      _stMsg.eType                  := E_MessageType.eMessageError;
      _stMsg.eDevice                := e_Device.Axis + TO_DINT(_AxisRef.NcToPlc.AxisId);
      _stMsg.eSubdevice             := e_Subdevice.fbCoeRead;

      _stMsg.iErrorNumber           := SEL((_fbCoeRead.CANopenErrId > 0), _fbCoeRead.AdsErrId, _fbCoeRead.CANopenErrId);

      _stMsg.sText                  := TO_STRING(_eState);
      f_MessageSet(_stMsg);

      _fbCoeRead(
                Execute             := FALSE,
                NetId               := _AxisRef.ADS.NetId, 
                Axis                := _AxisRef);

    ELSIF NOT _fbCoeRead.Busy
    THEN
      _eState                       := E_PROGRESS.WORKING;
    END_IF
*)
END_CASE
CASE _eState
OF
  E_PROGRESS.PROGRESS_WORKING:
    _eState                         := E_PROGRESS.PROGRESS_DONE;
    // set default for axis release
    AxisEnableNegative              := TRUE;
    AxisEnablePositive              := TRUE;

    // clear fb
    _fbCoeRead(
              Execute               := FALSE,
              NetId                 := _AxisRef.ADS.NetId, 
              Axis                  := _AxisRef);

    _stMsg.eType                    := E_MessageType.eMessageInfo;
    _stMsg.eDevice                  := e_Device.Axis + (_AxisRef.NcToPlc.AxisId);
    _stMsg.eSubdevice               := e_Subdevice.AxisStartUp;
    _stMsg.iErrorNumber             := 0;
    _stMsg.sText                    := concat('Axis Init: ', _sDeviceName);
    _stMsg.sText                    := concat(_stMsg.sText, ' : ');
    _stMsg.sText                    := concat(_stMsg.sText, TO_STRING(_eState));

  IF (_MessageLevel > E_MessageType.eMessageError)
  THEN
    f_MessageSet(_stMsg);
  END_IF
END_CASE

AxisInit                            := _eState;
END_METHOD

METHOD AxisMoveToPosition : E_PROGRESS
VAR_INPUT
  Execute           : BOOL;
  Data              : ST_MOVE_DATA;
END_VAR
VAR_INST
  _eres,
  _eState           : E_PROGRESS;
END_VAR
IF NOT Check() THEN AxisMoveToPosition := E_PROGRESS.PROGRESS_ERROR; RETURN; END_IF
IF NOT Execute THEN _eState := E_PROGRESS.PROGRESS_INIT; END_IF

CASE _eState
OF
  E_PROGRESS.PROGRESS_INIT:
    IF Execute 
    THEN
      _eState               := E_PROGRESS.PROGRESS_BUSY;
    END_IF
END_CASE
CASE _eState
OF
  E_PROGRESS.PROGRESS_BUSY:
    _eState                 := E_PROGRESS.PROGRESS_OCCUPIED;
    _eres                   := MoveToPos(
                                      Execute    := FALSE, 
                                      Position   := Data.rSetPos, 
                                      Vel        := Data.rSetVelo, 
                                      Acc        := Data.rAcc, 
                                      Dec        := Data.rDec, 
                                      Jerk       := Data.rJerk, 
                                      BufferMode := Tc2_MC2.MC_BufferMode.MC_Aborting);
END_CASE
CASE _eState
OF
  E_PROGRESS.PROGRESS_OCCUPIED:
    _eres                   := MoveToPos(
                                      Execute    := TRUE, 
                                      Position   := Data.rSetPos, 
                                      Vel        := Data.rSetVelo, 
                                      Acc        := Data.rAcc, 
                                      Dec        := Data.rDec, 
                                      Jerk       := Data.rJerk, 
                                      BufferMode := Tc2_MC2.MC_BufferMode.MC_Aborting);

    IF (_eres = E_PROGRESS.PROGRESS_ERROR)
    THEN
        _eState             := E_PROGRESS.PROGRESS_ERROR;
    ELSIF (_eres = E_PROGRESS.PROGRESS_DONE)
    THEN 
      _eState               := E_PROGRESS.PROGRESS_WORKING;
    END_IF
END_CASE
CASE _eState
OF
  E_PROGRESS.PROGRESS_WORKING:
    _eState                 := E_PROGRESS.PROGRESS_DONE;
    _eres                   := MoveToPos(
                                      Execute    := FALSE, 
                                      Position   := Data.rSetPos, 
                                      Vel        := Data.rSetVelo, 
                                      Acc        := Data.rAcc, 
                                      Dec        := Data.rDec, 
                                      Jerk       := Data.rJerk, 
                                      BufferMode := Tc2_MC2.MC_BufferMode.MC_Aborting);
END_CASE

AxisMoveToPosition := _eState;
END_METHOD

METHOD AxisMoveVelocity : E_PROGRESS
VAR_INPUT
  Execute           : BOOL;
  Data              : ST_MOVE_DATA;
END_VAR
VAR_INST
  _eres,
  _eState           : E_PROGRESS;
END_VAR
IF NOT Check() THEN AxisMoveVelocity := E_PROGRESS.PROGRESS_ERROR; RETURN; END_IF
IF NOT Execute THEN _eState := E_PROGRESS.PROGRESS_INIT; END_IF

CASE _eState
OF
  E_PROGRESS.PROGRESS_INIT:
    IF Execute 
    THEN
      _eState               := E_PROGRESS.PROGRESS_BUSY;
    END_IF
END_CASE
CASE _eState
OF
  E_PROGRESS.PROGRESS_BUSY:
    _eState                 := E_PROGRESS.PROGRESS_OCCUPIED;
    _eres                   := MoveVelo(
                                    Execute     := FALSE, 
                                    Velocity    := Data.rSetVelo, 
                                    Acc         := Data.rAcc, 
                                    Dec         := Data.rDec, 
                                    Jerk        := Data.rJerk, 
                                    Direction   := Data.iDirection, 
                                    BufferMode  := Tc2_MC2.MC_BufferMode.MC_Aborting);
END_CASE
CASE _eState
OF
  E_PROGRESS.PROGRESS_OCCUPIED:
    _eres                   := MoveVelo(
                                    Execute     := TRUE, 
                                    Velocity    := Data.rSetVelo, 
                                    Acc         := Data.rAcc, 
                                    Dec         := Data.rDec, 
                                    Jerk        := Data.rJerk, 
                                    Direction   := Data.iDirection, 
                                    BufferMode  := Tc2_MC2.MC_BufferMode.MC_Aborting);
    IF (_eres = E_PROGRESS.PROGRESS_ERROR)
    THEN
        _eState             := E_PROGRESS.PROGRESS_ERROR;
    ELSIF (_eres = E_PROGRESS.PROGRESS_DONE)
    THEN 
      _eState               := E_PROGRESS.PROGRESS_WORKING;
    END_IF
END_CASE
CASE _eState
OF
  E_PROGRESS.PROGRESS_WORKING:
    _eState                 := E_PROGRESS.PROGRESS_DONE;
    _eres                   := MoveVelo(
                                    Execute     := FALSE, 
                                    Velocity    := Data.rSetVelo, 
                                    Acc         := Data.rAcc, 
                                    Dec         := Data.rDec, 
                                    Jerk        := Data.rJerk, 
                                    Direction   := Data.iDirection, 
                                    BufferMode  := Tc2_MC2.MC_BufferMode.MC_Aborting);
END_CASE

AxisMoveVelocity                := _eState;
END_METHOD

METHOD AxisParameterRead : E_PROGRESS
VAR_INPUT
  Execute           : BOOL;
  ParameterNr       : Tc2_MC2.MC_AxisParameter;
END_VAR
VAR_INST
  _eres,
  _eState           : E_PROGRESS;
  _rValue           : LREAL;
END_VAR
IF NOT Check() THEN AxisParameterRead := E_PROGRESS.PROGRESS_ERROR; RETURN; END_IF
IF NOT Execute THEN _eState := E_PROGRESS.PROGRESS_INIT; END_IF

CASE _eState
OF
  E_PROGRESS.PROGRESS_INIT:
    IF Execute 
    THEN
      _rValue                                     := 0.0;
      _eState                                     := E_PROGRESS.PROGRESS_BUSY;
    END_IF
END_CASE
CASE _eState
OF
  E_PROGRESS.PROGRESS_BUSY:
    _eState                                       := E_PROGRESS.PROGRESS_OCCUPIED;
    _eres           := ReadParameter(
                                  Execute         := FALSE,
                                  ParameterNumber := ParameterNr);
END_CASE
CASE _eState
OF
  E_PROGRESS.PROGRESS_OCCUPIED:
    _eres           := ReadParameter(
                                  Execute         := TRUE,
                                  ParameterNumber := ParameterNr);

    IF (_eres = E_PROGRESS.PROGRESS_ERROR)
    THEN
      _eState                                     := E_PROGRESS.PROGRESS_ERROR;
    ELSIF (_eres = E_PROGRESS.PROGRESS_DONE)
    THEN 
      _eState                                     := E_PROGRESS.PROGRESS_WORKING;
    END_IF

  E_PROGRESS.PROGRESS_WORKING:
    _eState                                       := E_PROGRESS.PROGRESS_DONE;
    _eres           := ReadParameter(
                                  Execute         := FALSE,
                                  ParameterNumber := ParameterNr);

    _NcParameterWrt^[_nAxisIndex].rValue          :=
    _rParameterReadValue                          := 
    _rValue                                       :=ReadParameterValue;
END_CASE

AxisParameterRead := _eState;
END_METHOD

METHOD AxisParameterWrite : E_PROGRESS
VAR_INPUT
  Execute           : BOOL;
  ParameterNr       : Tc2_MC2.MC_AxisParameter;
END_VAR
VAR_INST
  _eres,
  _eState           : E_PROGRESS;
  _rValue           : LREAL;
END_VAR
IF NOT Check() THEN AxisParameterWrite := E_PROGRESS.PROGRESS_ERROR; RETURN; END_IF
IF NOT Execute THEN _eState := E_PROGRESS.PROGRESS_INIT; END_IF

CASE _eState
OF
  E_PROGRESS.PROGRESS_INIT:
    IF Execute 
    THEN
      _rValue                                     := _NcParameterWrt^[_nAxisIndex].rValue;
      _eState                                     := E_PROGRESS.PROGRESS_BUSY;
    END_IF
END_CASE
CASE _eState
OF
  E_PROGRESS.PROGRESS_BUSY:
    _eState                                       := E_PROGRESS.PROGRESS_OCCUPIED;
    _eres           := WriteParameter(
                                  Execute         := FALSE,
                                  Value           := _rValue,
                                  ParameterNumber := ParameterNr);
END_CASE
CASE _eState
OF
  E_PROGRESS.PROGRESS_OCCUPIED:
    _eres           := WriteParameter(
                                  Execute         := TRUE,
                                  Value           := _rValue,
                                  ParameterNumber := ParameterNr);
    IF (_eres = E_PROGRESS.PROGRESS_ERROR)
    THEN
      _eState                                     := E_PROGRESS.PROGRESS_ERROR;
    ELSIF (_eres = E_PROGRESS.PROGRESS_DONE)
    THEN 
      _eState                                     := E_PROGRESS.PROGRESS_WORKING;
    END_IF

  E_PROGRESS.PROGRESS_WORKING:
    _eState                                       := E_PROGRESS.PROGRESS_DONE;
    _eres           := WriteParameter(
                                  Execute         := FALSE,
                                  Value           := _rValue,
                                  ParameterNumber := ParameterNr);
END_CASE

AxisParameterWrite                                    := _eState;
END_METHOD

METHOD AxisParameterWritePersistent : E_PROGRESS
VAR_INPUT
  Execute           : BOOL;
  ParameterNr       : Tc2_MC2.MC_AxisParameter;
END_VAR
VAR_INST
  _eres,
  _eState           : E_PROGRESS;
  _rValue           : LREAL;
END_VAR
IF NOT Check() THEN AxisParameterWritePersistent := E_PROGRESS.PROGRESS_ERROR; RETURN; END_IF
IF NOT Execute THEN _eState := E_PROGRESS.PROGRESS_INIT; END_IF

CASE _eState
OF
  E_PROGRESS.PROGRESS_INIT:
    IF Execute 
    THEN
      _rValue                                     := _NcParameterWrt^[_nAxisIndex].rValue;
      _eState                                     := E_PROGRESS.PROGRESS_BUSY;
    END_IF
END_CASE
CASE _eState
OF
  E_PROGRESS.PROGRESS_BUSY:
    _eState                                       := E_PROGRESS.PROGRESS_OCCUPIED;
    _eres           := WriteParameterPersistent(
                                  Execute         := FALSE,
                                  Value           := _rValue,
                                  ParameterNumber := ParameterNr);
END_CASE
CASE _eState
OF
  E_PROGRESS.PROGRESS_OCCUPIED:
    _eres           := WriteParameterPersistent(
                                  Execute         := TRUE,
                                  Value           := _rValue,
                                  ParameterNumber := ParameterNr);
    IF (_eres = E_PROGRESS.PROGRESS_ERROR)
    THEN
      _eState                                     := E_PROGRESS.PROGRESS_ERROR;
    ELSIF (_eres = E_PROGRESS.PROGRESS_DONE)
    THEN 
      _eState                                     := E_PROGRESS.PROGRESS_WORKING;
    END_IF

  E_PROGRESS.PROGRESS_WORKING:
    _eState                                       := E_PROGRESS.PROGRESS_DONE;
    _eres           := WriteParameterPersistent(
                                  Execute         := FALSE,
                                  Value           := _rValue,
                                  ParameterNumber := ParameterNr);
END_CASE

AxisParameterWritePersistent                          := _eState;
END_METHOD

METHOD AxisReset : E_PROGRESS
VAR_INPUT
  Execute           : BOOL;
END_VAR
VAR_INST
  _eres,
  _eState           : E_PROGRESS;
END_VAR
IF NOT Check() THEN AxisReset := E_PROGRESS.PROGRESS_ERROR; RETURN; END_IF
IF NOT Execute THEN _eState := E_PROGRESS.PROGRESS_INIT; END_IF

CASE _eState
OF
  E_PROGRESS.PROGRESS_INIT:
    IF Execute 
    THEN
      _eState                       := E_PROGRESS.PROGRESS_BUSY;
    END_IF
END_CASE
CASE _eState
OF
  E_PROGRESS.PROGRESS_BUSY:
    _eres                           := Reset(FALSE);
    _eState                         := E_PROGRESS.PROGRESS_OCCUPIED;
END_CASE
CASE _eState
OF
  E_PROGRESS.PROGRESS_OCCUPIED:
    _eres                           := Reset(TRUE);
    IF (_eres = E_PROGRESS.PROGRESS_DONE)
    THEN
      _eState                       := E_PROGRESS.PROGRESS_WORKING;
    ELSIF (_eres = E_PROGRESS.PROGRESS_ERROR)
    THEN
      _eState                       := E_PROGRESS.PROGRESS_ERROR;
    END_IF
END_CASE
CASE _eState
OF
  E_PROGRESS.PROGRESS_WORKING:
    _eres                           := Reset(FALSE);
    _eState                         := E_PROGRESS.PROGRESS_DONE;
END_CASE

AxisReset                           := _eState;
END_METHOD

METHOD AxisSendToPosition : E_PROGRESS
VAR_INPUT
  Execute           : BOOL;
  Data              : ST_MOVE_DATA;
END_VAR
VAR_INST
  _eres,
  _eState           : E_PROGRESS;
END_VAR
IF NOT Check() THEN AxisSendToPosition := E_PROGRESS.PROGRESS_ERROR; RETURN; END_IF
IF NOT Execute THEN _eState := E_PROGRESS.PROGRESS_INIT; END_IF

CASE _eState
OF
  E_PROGRESS.PROGRESS_INIT:
    IF Execute 
    THEN
      _eState               := E_PROGRESS.PROGRESS_BUSY;
    END_IF
END_CASE
CASE _eState
OF
  E_PROGRESS.PROGRESS_BUSY:
    _eState                 := E_PROGRESS.PROGRESS_OCCUPIED;
    _eres                   := SendToPos(
                                      Execute    := FALSE, 
                                      Position   := Data.rSetPos, 
	                                    Distance   := _MotionOptions^[_nAxisIndex].rDistance, 
                                      Vel        := Data.rSetVelo, 
                                      Acc        := Data.rAcc, 
                                      Dec        := Data.rDec, 
                                      Jerk       := Data.rJerk, 
	                                    BufferMode := Tc2_MC2.MC_BufferMode.MC_Aborting);
END_CASE
CASE _eState
OF
  E_PROGRESS.PROGRESS_OCCUPIED:
    _eres                   := SendToPos(
                                      Execute    := TRUE, 
                                      Position   := Data.rSetPos, 
	                                    Distance   := _MotionOptions^[_nAxisIndex].rDistance, 
                                      Vel        := Data.rSetVelo, 
                                      Acc        := Data.rAcc, 
                                      Dec        := Data.rDec, 
                                      Jerk       := Data.rJerk, 
	                                    BufferMode := Tc2_MC2.MC_BufferMode.MC_Aborting);

    IF (_eres = E_PROGRESS.PROGRESS_ERROR)
    THEN
        _eState             := E_PROGRESS.PROGRESS_ERROR;
    ELSIF (_eres = E_PROGRESS.PROGRESS_DONE)
    THEN 
      _eState               := E_PROGRESS.PROGRESS_WORKING;
    END_IF
END_CASE
CASE _eState
OF
  E_PROGRESS.PROGRESS_WORKING:
    _eState                 := E_PROGRESS.PROGRESS_DONE;
    _eres                   := SendToPos(
                                      Execute    := FALSE, 
                                      Position   := Data.rSetPos, 
	                                    Distance   := _MotionOptions^[_nAxisIndex].rDistance, 
                                      Vel        := Data.rSetVelo, 
                                      Acc        := Data.rAcc, 
                                      Dec        := Data.rDec, 
                                      Jerk       := Data.rJerk, 
	                                    BufferMode := Tc2_MC2.MC_BufferMode.MC_Aborting);
END_CASE

AxisSendToPosition := _eState;
END_METHOD

PROPERTY AxisState : pointer to ARRAY[1..PLC_CONSTANT.MAX_AXIS] OF ST_AXIS_STATE
SET
_State := AxisState;
END_SET
END_PROPERTY

METHOD AxisStop : E_PROGRESS
VAR_INPUT
  Execute           : BOOL;
  Data              : ST_MOVE_DATA;
END_VAR
VAR_INST
  _eres,
  _eState           : E_PROGRESS;
END_VAR
IF NOT Check() THEN AxisStop := E_PROGRESS.PROGRESS_ERROR; RETURN; END_IF
IF NOT Execute THEN _eState := E_PROGRESS.PROGRESS_INIT; END_IF

CASE _eState
OF
  E_PROGRESS.PROGRESS_INIT:
    IF Execute 
    THEN
      _eState       := E_PROGRESS.PROGRESS_BUSY;
    END_IF
END_CASE
CASE _eState
OF
  E_PROGRESS.PROGRESS_BUSY:
    _eState         := E_PROGRESS.PROGRESS_OCCUPIED;
    _eres           := Stop(
                            Execute := FALSE, 
                            Dec     := Data.rDec, 
                            Jerk    := Data.rJerk);
END_CASE
CASE _eState
OF
  E_PROGRESS.PROGRESS_OCCUPIED:
    _eres           := Stop(
                            Execute := TRUE, 
                            Dec     := Data.rDec, 
                            Jerk    := Data.rJerk);

    IF (_eres = E_PROGRESS.PROGRESS_ERROR)
    THEN
        _eState     := E_PROGRESS.PROGRESS_ERROR;
    ELSIF (_eres = E_PROGRESS.PROGRESS_DONE)
    THEN 
      _eState       := E_PROGRESS.PROGRESS_WORKING;
    END_IF
END_CASE
CASE _eState
OF
  E_PROGRESS.PROGRESS_WORKING:
    _eState         := E_PROGRESS.PROGRESS_DONE;
    _eres           := Stop(
                            Execute := FALSE, 
                            Dec     := Data.rDec, 
                            Jerk    := Data.rJerk);
END_CASE

AxisStop := _eState;
END_METHOD

METHOD PRIVATE Check : BOOL
//-----------------------------------------------------------------------------
IF (_nAxisIndex < 1) OR
   (_nAxisIndex > PLC_CONSTANT.MAX_AXIS)
THEN
  _eCheck                 := E_CHECK_STATE.AXIS_INDEX_OUT_OF_RANGE;
  RETURN;
END_IF

IF NOT __ISVALIDREF(_Axes)
THEN
  _eCheck                 := E_CHECK_STATE.AXIS_REF_POINTER_INVALID;
  RETURN;
END_IF
//-----------------------------------------------------------------------------
// get my AXIS_REF pointer for use in base class
//-----------------------------------------------------------------------------
_AxisRef                  := _Axes[_nAxisIndex];
//-----------------------------------------------------------------------------

IF NOT (_Ctrl <> 0)
THEN
  _eCheck                 := E_CHECK_STATE.AXIS_CTRL_POINTER_INVALID;
  RETURN;
END_IF

IF NOT (_State <> 0)
THEN
  _eCheck                 := E_CHECK_STATE.AXIS_STATE_POINTER_INVALID;
  RETURN;
END_IF

IF NOT (_Info <> 0)
THEN
  _eCheck                 := E_CHECK_STATE.AXIS_INFO_POINTER_INVALID;
  RETURN;
END_IF

IF NOT (_Data <> 0)
THEN
  _eCheck                 := E_CHECK_STATE.AXIS_DATA_POINTER_INVALID;
  RETURN;
END_IF

IF NOT (_NcParameterWrt <> 0)
THEN
  _eCheck                 := E_CHECK_STATE.AXIS_NC_PARAMETER_POINTER_INVALID;
  RETURN;
END_IF

IF NOT (_NcParameterRd <> 0)
THEN
  _eCheck                 := E_CHECK_STATE.AXIS_NC_PARAMETER_POINTER_INVALID;
  RETURN;
END_IF

IF NOT (_HomeParameter <> 0)
THEN
  _eCheck                 := E_CHECK_STATE.AXIS_HOME_PARAMETER_POINTER_INVALID;
  RETURN;
END_IF

IF NOT (_GearInParameter <> 0)
THEN
  _eCheck                 := E_CHECK_STATE.AXIS_GEAR_IN_PARAMETER_POINTER_INVALID;
  RETURN;
END_IF
  
IF NOT (_MotionOptions <> 0)
THEN
  _eCheck                 := E_CHECK_STATE.AXIS_MOTION_OPTIONS_POINTER_INVALID;
  RETURN;
END_IF

//-----------------------------------------------------------------------------
//  NaN INF check
//-----------------------------------------------------------------------------
IF NOT IsFinite(F_LReal(_Data^[_nAxisIndex].rSetPos))
THEN
	_Data^[_nAxisIndex].rSetPos     := 0.0;
END_IF

IF NOT IsFinite(F_LReal(_Data^[_nAxisIndex].rSetVelo))
THEN
	_Data^[_nAxisIndex].rSetVelo    := 0.0;
END_IF

IF NOT IsFinite(F_LReal(_Data^[_nAxisIndex].rAcc))
THEN
	_Data^[_nAxisIndex].rAcc        := 0.0;
END_IF

IF NOT IsFinite(F_LReal(_Data^[_nAxisIndex].rDec))
THEN
	_Data^[_nAxisIndex].rDec        := 0.0;
END_IF

IF NOT IsFinite(F_LReal(_Data^[_nAxisIndex].rOverride))
THEN
	_Data^[_nAxisIndex].rOverride   := 0.0;
END_IF
//-----------------------------------------------------------------------------
//-----------------------------------------------------------------------------
_eCheck                   := E_CHECK_STATE.CHECK_DONE;
Check                     := TRUE;
//-----------------------------------------------------------------------------
//-----------------------------------------------------------------------------
END_METHOD

//-------------------------------------------------------------------------------------
//
//  HAUD 2024 01 20
//
//  Cmd
//    - gets state for ctrl
//    - checks for eInit to be done, before any other commands are accepted
//    - prepare your commands here
//    - init what you have to here
//
//-------------------------------------------------------------------------------------
METHOD PRIVATE Cmd  : E_AXIS_STATE
VAR_INPUT
  eCmd              : E_AXIS_CTRL;
END_VAR
VAR_INST
  _estate   : E_AXIS_STATE;
  _stMsg    : ST_Message;
END_VAR

CASE eCmd
OF
  //-------------------------------------------------------------------------------------
  E_AXIS_CTRL.AXIS_INIT:
    _eInit    := _eResult             := AxisInit(FALSE);
    _estate                           := E_AXIS_STATE.AXIS_INIT;
ELSE
  IF (_eInit <> E_PROGRESS.PROGRESS_DONE)
  THEN
    _eResult                          := E_PROGRESS.PROGRESS_INIT;
    _estate                           := E_AXIS_STATE.AXIS_NO_INIT;
  ELSE
    CASE eCmd
    OF
      //---------------------------------------------------------------------------------
      E_AXIS_CTRL.AXIS_DISABLE:
        _eResult                      := AxisDisable(FALSE);
        _estate                       := E_AXIS_STATE.AXIS_DISABLE;

      //---------------------------------------------------------------------------------
      E_AXIS_CTRL.AXIS_ENABLE:
        _eResult                      := AxisEnable(FALSE);
        _estate                       := E_AXIS_STATE.AXIS_ENABLE;

      //---------------------------------------------------------------------------------
      E_AXIS_CTRL.AXIS_IDLE:
        _eResult                      := AxisBufferVelo(FALSE, _Data^[_nAxisIndex]);
        _eResult                      := AxisBufferPos(FALSE, _Data^[_nAxisIndex]);
        _eResult                      := AxisIdle(FALSE);
        _estate                       := E_AXIS_STATE.AXIS_IDLE;

      //---------------------------------------------------------------------------------
      E_AXIS_CTRL.AXIS_HOME:
        _eResult                      := AxisHome(FALSE);
        _estate                       := E_AXIS_STATE.AXIS_HOME;

      //---------------------------------------------------------------------------------
      E_AXIS_CTRL.AXIS_MOVE_POS:
        _eResult                      := AxisMoveToPosition(FALSE, _Data^[_nAxisIndex]);
        _estate                       := E_AXIS_STATE.AXIS_MOVE_POS;

      //---------------------------------------------------------------------------------
      E_AXIS_CTRL.AXIS_MOVE_VELO:
        _eResult                      := AxisMoveVelocity(FALSE, _Data^[_nAxisIndex]);
        _estate                       := E_AXIS_STATE.AXIS_MOVE_VELO;

      E_AXIS_CTRL.AXIS_SEND_TO_POS:
        _eResult                      := AxisSendToPosition(FALSE, _Data^[_nAxisIndex]);
        _estate                       := E_AXIS_STATE.AXIS_SEND_TO_POS;

      //---------------------------------------------------------------------------------
      E_AXIS_CTRL.AXIS_RESET:
        // OnChange clear error bit
        _Info^[_nAxisIndex].bError    := FALSE;
        _eResult                      := AxisReset(FALSE);
        _estate                       := E_AXIS_STATE.AXIS_RESET;

      //---------------------------------------------------------------------------------
      E_AXIS_CTRL.AXIS_HALT:
        _eResult                      := AxisHalt(FALSE, _Data^[_nAxisIndex]);
        _estate                       := E_AXIS_STATE.AXIS_HALT;

      //---------------------------------------------------------------------------------
      E_AXIS_CTRL.AXIS_STOP:
        _eResult                      := AxisStop(FALSE, _Data^[_nAxisIndex]);
        _estate                       := E_AXIS_STATE.AXIS_STOP;


      //---------------------------------------------------------------------------------
      E_AXIS_CTRL.AXIS_MOVE_BUFFER:
        _eResult                      := AxisBufferPos(FALSE, _Data^[_nAxisIndex]);
        _estate                       := E_AXIS_STATE.AXIS_MOVE_BUFFER;


      //---------------------------------------------------------------------------------
      E_AXIS_CTRL.AXIS_MOVE_BUFFER_VELO:
        _eResult                      := AxisBufferVelo(FALSE, _Data^[_nAxisIndex]);
        _estate                       := E_AXIS_STATE.AXIS_MOVE_BUFFER_VELO;


      //---------------------------------------------------------------------------------
      E_AXIS_CTRL.AXIS_PARAMETER_READ:
        _eParameterNrRead             := _NcParameterRd^[_nAxisIndex].ParameterNumber;
        _eResult                      := AxisParameterRead(FALSE, _eParameterNrRead);
        _estate                       := E_AXIS_STATE.AXIS_PARAMETER_READ;


      //---------------------------------------------------------------------------------
      E_AXIS_CTRL.AXIS_PARAMETER_WRITE:
        _eParameterNrWrite            := _NcParameterWrt^[_nAxisIndex].ParameterNumber;
        _rParameterWrtValue           := _NcParameterWrt^[_nAxisIndex].rValue;
        _eResult                      := AxisParameterWrite(FALSE, _eParameterNrWrite);
        _estate                       := E_AXIS_STATE.AXIS_PARAMETER_WRITE;


      //---------------------------------------------------------------------------------
      E_AXIS_CTRL.AXIS_PARAMETER_WRITE_PERSISTENT:
        _eParameterNrWrite            := _NcParameterWrt^[_nAxisIndex].ParameterNumber;
        _rParameterWrtValue           := _NcParameterWrt^[_nAxisIndex].rValue;
        _eResult                      := AxisParameterWritePersistent(FALSE, _eParameterNrWrite);
        _estate                       := E_AXIS_STATE.AXIS_PARAMETER_WRITE_PERSISTENT;

      //---------------------------------------------------------------------------------
      E_AXIS_CTRL.AXIS_GEAR_IN:
        _eResult                      := AxisGearIn(FALSE);
        _estate                       := E_AXIS_STATE.AXIS_GEAR_IN;

      //---------------------------------------------------------------------------------    
      E_AXIS_CTRL.AXIS_GEAR_OUT:
        _eResult                      := AxisGearOut(FALSE);
        _estate                       := E_AXIS_STATE.AXIS_GEAR_OUT;

      //---------------------------------------------------------------------------------
      E_AXIS_CTRL.AXIS_GEAR_IN_MULTIMASTER:
        _fbGearInMultiMaster.Master1  := _MultiMasterDummyRef[1];
        _fbGearInMultiMaster.Master2  := _MultiMasterDummyRef[2];
        _fbGearInMultiMaster.Master3  := _MultiMasterDummyRef[3];
        _fbGearInMultiMaster.Master4  := _MultiMasterDummyRef[4];

        _eResult                      := AxisGearInMultiMaster(FALSE);
        _estate                       := E_AXIS_STATE.AXIS_GEAR_IN_MULTIMASTER;

    //-----------------------------------------------------------------------------------
    ELSE
      _estate                         := E_AXIS_STATE.AXIS_NULL;

      IF (eCmd = E_AXIS_CTRL.AXIS_NULL)
      THEN
        _eResult                      := E_PROGRESS.PROGRESS_DONE;
      ELSE
        _eResult                      := E_PROGRESS.PROGRESS_INVALID;
  
        _stMsg.eType                  := E_MessageType.eMessageError;
        _stMsg.eDevice                := E_Device.Axis + (_Axes[_nAxisIndex].NcToPlc.AxisId);
        _stMsg.eSubdevice             := e_Subdevice.AxisControl;
        _stMsg.iErrorNumber           := 0;
  
        _stMsg.sText                  := 'E_AXIS_CTRL.';
        _stMsg.sText                  := concat(_stMsg.sText, TO_STRING(eCmd));
        _stMsg.sText                  := concat(_stMsg.sText, ': ');
        _stMsg.sText                  := concat(_stMsg.sText, TO_STRING(_eResult));

        f_MessageSet(_stMsg);
      END_IF
    END_CASE
  END_IF // _eInit
END_CASE

Cmd                                   := _estate;
END_METHOD

METHOD PRIVATE GetCalibrationCam : BOOL
VAR_INST
  _bCal     : Bool;
END_VAR
IF NOT Check() THEN RETURN; END_IF

IF _HomeParameter^[_nAxisIndex].stHomingParam.SimulateHomeSensor
THEN
	IF (_AxisRef.NcToPlc.HomingState < 4)
  THEN
		_bCal := TRUE;
	ELSE
		_bCal := FALSE;
	END_IF
ELSIF _HomeParameter^[_nAxisIndex].stHomingParam.HomeOnLimitMin
THEN
	_bCal := _bLimitMin XOR _HomeParameter^[_nAxisIndex].stHomingParam.InvertHomeSensor;

ELSIF _HomeParameter^[_nAxisIndex].stHomingParam.HomeOnLimitMax
THEN
	_bCal := _bLimitMax XOR _HomeParameter^[_nAxisIndex].stHomingParam.InvertHomeSensor;
ELSE
	_bCal := _bCalibrationInput XOR _HomeParameter^[_nAxisIndex].stHomingParam.InvertHomeSensor;
END_IF

GetCalibrationCam := _bCal;
END_METHOD

PROPERTY HomingParameter : pointer to ARRAY[1..PLC_CONSTANT.MAX_AXIS] OF st_homing
SET
_HomeParameter := HomingParameter;
END_SET
END_PROPERTY

METHOD PRIVATE LogControl
VAR_INST
  _sResult,
  _sCtrl            : STRING(30);

  _stMsg            : ST_Message;
END_VAR
  _stMsg.eType               := E_MessageType.eMessageInfo;
  _stMsg.eDevice             := E_Device.Axis + (_AxisRef.NcToPlc.AxisId);
  _stMsg.eSubdevice          := e_Subdevice.AxisControl;
  _stMsg.iErrorNumber        := _nAxisIndex;

  _sCtrl                     := concat('E_AXIS_CTRL', '.');
  _sCtrl                     := concat(_sCtrl, TO_STRING(_eCmd));

  _stMsg.sText               := concat('new command: ', _sCtrl);

  IF (_MessageLevel > E_MessageType.eMessageError)
  THEN
    f_MessageSet(_stMsg);
  END_IF
END_METHOD

METHOD PRIVATE LogResult
VAR_INST
  _sResult,
  _sCtrl            : STRING(30);

  _stMsg            : ST_Message;
END_VAR

  _stMsg.eType               := E_MessageType.eMessageInfo;
  _stMsg.eDevice             := E_Device.Axis + (_AxisRef.NcToPlc.AxisId);
  _stMsg.eSubdevice          := e_Subdevice.AxisControl;
  _stMsg.iErrorNumber        := _nAxisIndex;

  _sCtrl                     := concat('E_AXIS_CTRL', '.');
  _sCtrl                     := concat(_sCtrl, TO_STRING(_eCmd));

  _sResult                   := concat('E_PROGRESS', '.');
  _sResult                   := concat(_sResult, TO_STRING(_eResult));

  _stMsg.sText               := concat(_sCtrl, ' ');
  _stMsg.sText               := concat(_sCtrl, _sResult);

  IF (_MessageLevel > E_MessageType.eMessageError)
  THEN
    f_MessageSet(_stMsg);
  END_IF
END_METHOD

PROPERTY MotionOptions : pointer to ARRAY[1..PLC_CONSTANT.MAX_AXIS] OF ST_MOTION_OPTIONS
SET
_MotionOptions := MotionOptions;
END_SET
END_PROPERTY

PROPERTY NcParameterValue : Lreal
GET
NcParameterValue := _rParameterReadValue;
END_GET
END_PROPERTY

PROPERTY ReadNcParameter : pointer to ARRAY[1..PLC_CONSTANT.MAX_AXIS] OF st_nc_parameter
SET
_NcParameterRd := ReadNcParameter;
END_SET
END_PROPERTY

METHOD PRIVATE ResetSoE : E_PROGRESS
VAR_INPUT
  Execute           : BOOL;
END_VAR
VAR_INST
  _eState           : E_PROGRESS;
  _rValue           : LREAL;
  _udiErrSer,
  _udiErrAds        : UDINT;
  _stMsg            : ST_Message;

	_fbReset		      : Tc2_MC2_Drive.FB_SoEReset;
  _tonDelay         : Tc2_Standard.TON;
	_nRepeat			    : UINT;

  _sErrorSercos     : Tc2_System.T_MaxString;

END_VAR
IF NOT Check() THEN ResetSoE := E_PROGRESS.PROGRESS_ERROR; RETURN; END_IF
IF NOT Execute THEN _eState := E_PROGRESS.PROGRESS_INIT; END_IF

CASE _eState
OF
  E_PROGRESS.PROGRESS_INIT:
    IF Execute 
    THEN
      memset(ADR(_stMsg),0,SIZEOF(_stMsg));
      memset(ADR(_sErrorSercos),0,SIZEOF(_sErrorSercos));

		  _nRepeat                      := 1;
      _udiErrSer := _udiErrAds      := 0;
      _rValue                       := 0;
      _eState                       := E_PROGRESS.PROGRESS_BUSY;
    END_IF
END_CASE
CASE _eState
OF
  E_PROGRESS.PROGRESS_BUSY:
    _eState                         := E_PROGRESS.PROGRESS_OCCUPIED;
		_tonDelay(
            IN                      := FALSE);

		_fbReset(
            Execute                 := FALSE, 
            Timeout                 := T#2500MS, 
            Axis                    := _AxisRef);
END_CASE
CASE _eState
OF
  E_PROGRESS.PROGRESS_OCCUPIED:
		_tonDelay(
            PT                      := T#1500MS, 
            IN                      := TRUE);

		_fbReset(
            Execute                 := TRUE, 
            Axis                    := _AxisRef, 
            AdsErrId                => _udiErrAds, 
            SercosErrId             => _udiErrSer);

    IF _fbReset.Error
    THEN
      _stMsg.eType                  := E_MessageType.eMessageError;
      _stMsg.eDevice                := e_Device.Axis + (_AxisRef.NcToPlc.AxisId);
      _stMsg.eSubdevice             :=  e_SubDevice.fbResetSercos;
      _stMsg.iErrorNumber           := _udiErrAds;

      _sErrorSercos                 := Tc2_Utilities.DATA_TO_HEXSTR(ADR(_udiErrSer), SIZEOF(_udiErrSer), FALSE);

      _stMsg.sText                  := concat('Sercos Err Nr: ', _sErrorSercos);

      f_MessageSet(_stMsg);

      _Info^[_nAxisIndex].nErrorId := _udiErrSer;
      _eState                       := E_PROGRESS.PROGRESS_ERROR;

		ELSIF NOT _fbReset.Busy
		THEN
      _eState                       := E_PROGRESS.PROGRESS_WORKING;

    ELSE
      IF _tonDelay.Q AND
         _AxisRef.NcToPlc.StateDWord.28
      THEN
        _nRepeat                    := _nRepeat + 1;
        _eState                     := E_PROGRESS.PROGRESS_BUSY;    
      END_IF

      IF (_nRepeat > 5)
      THEN
        _eState                     := E_PROGRESS.PROGRESS_ERROR;
      END_IF
		END_IF
END_CASE
CASE _eState
OF
  E_PROGRESS.PROGRESS_WORKING:
    _eState                         := E_PROGRESS.PROGRESS_DONE;
END_CASE


ResetSoE := _eState;
END_METHOD

PROPERTY TargetWindow : lreal
GET
END_GET
SET
END_SET
END_PROPERTY

METHOD Template : E_PROGRESS
VAR_INPUT
  Execute           : BOOL;
END_VAR
VAR_INST
  _eState           : E_PROGRESS;
  _rValue           : LREAL;
  _udiErr           : UDINT;
  _stMsg            : ST_Message;


END_VAR
IF NOT Check() THEN _eState := E_PROGRESS.ERROR; END_IF
IF NOT Execute THEN _eState := E_PROGRESS.INIT; END_IF

CASE _eState
OF
  E_PROGRESS.INIT:
    IF Execute 
    THEN
      memset(ADR(_stMsg),0,SIZEOF(_stMsg));
      _udiErr                       := 0;
      _rValue                       := 0;
      _eState                       := E_PROGRESS.BUSY;
    END_IF
END_CASE
CASE _eState
OF
  E_PROGRESS.BUSY:
    _eState                         := E_PROGRESS.STARTUP;
END_CASE
CASE _eState
OF
  E_PROGRESS.STARTUP:
    _eState                         := E_PROGRESS.PREPARE;
END_CASE
CASE _eState
OF
  E_PROGRESS.PREPARE:
    _eState                         := E_PROGRESS.READY;
END_CASE
CASE _eState
OF
  E_PROGRESS.READY:
    _eState                         := E_PROGRESS.WAITING;
END_CASE
CASE _eState
OF
  E_PROGRESS.WAITING:
    _eState                         := E_PROGRESS.WORKING;
END_CASE
CASE _eState
OF
  E_PROGRESS.WORKING:
    _eState                         := E_PROGRESS.DONE;
END_CASE

Template_1 := _eState;
END_METHOD

PROPERTY WriteNcParameter : pointer to ARRAY[1..PLC_CONSTANT.MAX_AXIS] OF st_nc_parameter
SET
_NcParameterWrt := WriteNcParameter;
END_SET
END_PROPERTY

END_FUNCTION_BLOCK

// ---- NC_PTP/FB_McAxisBase.TcPOU
FUNCTION_BLOCK ABSTRACT FB_McAxisBase  IMPLEMENTS I_McAxis
VAR
  _AxisRef                      : REFERENCE TO Tc2_MC2.AXIS_REF;
  _pCalibrationCam              : POINTER TO BOOL;

  _nErrorId                     : UDINT; // datafield for MC error

  _MessageLevel                 : E_MessageType;

  // MC_Power inputs for feed fwd, feed bwd, override
  _bEnablePositive              : BOOL  := TRUE;
  _bEnableNegative              : BOOL  := TRUE;
  _rAxisOverride                : LREAL := 100.0;

  _rValueParameterRead          : LREAL;
  _fbReadParameter              : Tc2_MC2.MC_ReadParameter;
  _fbWriteParameter             : Tc2_MC2.MC_WriteParameter;
  _fbWriteParameterPersist      : Tc2_MC2.MC_WriteParameterPersistent;

  // last target position datafield
  _rLastTargetPosition          : LREAL;

  // name and encoder type are read by ADSREAD instance from NC
  _sAxisName                    : STRING(30) := 'NO NAME'; // AxisName is limited to 30 chars, IdxGrp := 4000 + _AxisRef.NcToPlc.AxisId, IdxOffs := 16#02
  _sEncoderType                 : STRING(30) := 'NO TYPE';
  _nEncoderType                 : UDINT;
  _eEncoderType                 : E_AxisEncoderType;

  // Motion Control FB Instances
  _fbPower                      : Tc2_MC2.MC_Power;
  _fbReset                      : Tc2_MC2.MC_Reset;
  _fbHalt                       : Tc2_MC2.MC_Halt;
  _fbStop                       : Tc2_MC2.MC_Stop;
  _fbHome                       : Tc2_MC2.MC_Home;
  _fbJog                        : Tc2_MC2.MC_Jog;
  _fbMoveToPosition             : Tc2_MC2.MC_MoveAbsolute;
  _fbMoveVelo                   : Tc2_MC2.MC_MoveVelocity;

  // used for buffered moves
  _fbMoveVelocity               : ARRAY[1..2]   OF  Tc2_MC2.MC_MoveVelocity;
  _fbMoveAbsolute               : ARRAY[1..2]   OF  Tc2_MC2.MC_MoveAbsolute;

  // ADS read instance for reading startup information from NC
  _fbADSRead                     : ADSREAD;

  // startup states for getting ADS information from NC
  _nStartUpErrorState,
  _nStartUp                     : DINT := 0;

  _bStartUpError,
  _bStartUp                     : BOOL;

  _rCycleTime                   : LREAL;
  _fbGetCurTaskIndex            : Tc2_System.GETCURTASKINDEX;
END_VAR

PROPERTY AxisEnableNegative : BOOL
GET
AxisEnableNegative := _bEnableNegative;
END_GET
SET
_bEnableNegative := AxisEnableNegative;
END_SET
END_PROPERTY

PROPERTY AxisEnablePositive : BOOL
GET
AxisEnablePositive  := _bEnablePositive;
END_GET
SET
_bEnablePositive := AxisEnablePositive;
END_SET
END_PROPERTY

PROPERTY AxisName : string(30)
GET
AxisName := _sAxisName;
END_GET
END_PROPERTY

PROPERTY AxisRef : reference to AXIS_REF
GET
AxisRef := _AxisRef;
END_GET
END_PROPERTY

PROPERTY CalibrationCam : pointer to bool
GET
CalibrationCam  := _pCalibrationCam;
END_GET
SET
_pCalibrationCam := CalibrationCam;
END_SET
END_PROPERTY

METHOD Cycle : E_PROGRESS
VAR_INST
  _eState           : E_PROGRESS;
  _rValue           : LREAL;
  _nErrorId         : UDINT;
  _stMsg            : ST_Message;
END_VAR
IF NOT (__ISVALIDREF(_AxisRef))
THEN
  Cycle                           := E_PROGRESS.PROGRESS_ERROR;
  RETURN;
END_IF

// call cyclic NC interface
_AxisRef();

_fbPower(
        Axis                      := _AxisRef, 
        Enable_Positive           := _bEnablePositive, 
        Enable_Negative           := _bEnableNegative, 
        Override                  := _rAxisOverride);

CASE _eState
OF
  E_PROGRESS.PROGRESS_INVALID:
    _fbGetCurTaskIndex();
    _rCycleTime                   := UDINT_TO_LREAL(_TaskInfo[_fbGetCurTaskIndex.index].CycleTime)/10000.0;

    _eState                       := E_PROGRESS.PROGRESS_BUSY;
END_CASE
CASE _eState
OF
  E_PROGRESS.PROGRESS_BUSY:
    IF (_fbPower.Error) OR
       (_AxisRef.Status.Error)
    THEN
      _eState                     := E_PROGRESS.PROGRESS_ERROR;

      _nErrorId                   := SEL((_fbPower.ErrorID > 0), _AxisRef.NcToPlc.ErrorCode, _fbPower.ErrorID);

      _stMsg.eType                := E_MessageType.eMessageError;
      _stMsg.eDevice              := e_Device.Axis + (_AxisRef.NcToPlc.AxisId);;
      _stMsg.eSubdevice           := e_Subdevice.AxisCycle;
      _stMsg.iErrorNumber         := _nErrorId;

      _stMsg.sText                  := concat(' : ', TO_STRING(_eState));

      f_MessageSet(_stMsg);
    ELSE
      _nErrorId                   := 0;
      _eState                     := E_PROGRESS.PROGRESS_WORKING;
    END_IF
END_CASE
CASE _eState
OF
  E_PROGRESS.PROGRESS_WORKING:
    // rinse, repeat
    _eState                       := E_PROGRESS.PROGRESS_BUSY;
    Cycle                         := E_PROGRESS.PROGRESS_WORKING;
END_CASE
CASE _eState
OF
  E_PROGRESS.PROGRESS_ERROR:
    IF NOT (_fbPower.Error)
    THEN
      _eState                     := E_PROGRESS.PROGRESS_BUSY;
    ELSE
      Cycle                       := E_PROGRESS.PROGRESS_ERROR;
    END_IF
END_CASE
END_METHOD

METHOD Disable : E_PROGRESS
VAR_INPUT
  Execute           : BOOL;
END_VAR
VAR_INST
  _eResult,
  _eState           : E_PROGRESS;
  _rValue           : LREAL;
  _stMsg            : ST_Message;
END_VAR
IF NOT (__ISVALIDREF(_AxisRef)) THEN  Disable  := E_PROGRESS.PROGRESS_ERROR; RETURN; END_IF
IF NOT Execute THEN _eState := E_PROGRESS.PROGRESS_INIT; END_IF

CASE _eState
OF
  E_PROGRESS.PROGRESS_INIT:
    IF Execute 
    THEN
      memset(ADR(_stMsg),0,SIZEOF(_stMsg));
      _nErrorId                     := 0;
      _rValue                       := 0;
      _eState                       := E_PROGRESS.PROGRESS_BUSY;
    END_IF
END_CASE
CASE _eState
OF
  E_PROGRESS.PROGRESS_BUSY:
    _fbPower.Enable                 := FALSE;
    _eResult                        := Reset(FALSE);
    _eState                         := E_PROGRESS.PROGRESS_STARTUP;

  E_PROGRESS.PROGRESS_STARTUP:
    IF _fbPower.Error OR
       _AxisRef.Status.Error
    THEN
      _eState                       := E_PROGRESS.PROGRESS_PREPARE;

      _stMsg.eType                  := E_MessageType.eMessageVerbose;
      _stMsg.eDevice                := E_Device.Axis + (_AxisRef.NcToPlc.AxisId);
      _stMsg.eSubdevice             := e_Subdevice.fbPower;
      _stMsg.iErrorNumber           := 0;

      _stMsg.sText                  := concat('clear error on disable : ', TO_STRING(_eState));

      IF (_MessageLevel = E_MessageType.eMessageVerbose)
      THEN
        f_MessageSet(_stMsg);
      END_IF
    ELSE
      _eState                       := E_PROGRESS.PROGRESS_OCCUPIED;
    END_IF
END_CASE
CASE _eState
OF
  E_PROGRESS.PROGRESS_PREPARE:
    _eResult                        := Reset(TRUE);
    IF (_eResult = E_PROGRESS.PROGRESS_DONE)
    THEN
      _eState                       := E_PROGRESS.PROGRESS_OCCUPIED;

      _stMsg.eType                  := E_MessageType.eMessageVerbose;
      _stMsg.eDevice                := E_Device.Axis + (_AxisRef.NcToPlc.AxisId);
      _stMsg.eSubdevice             := e_Subdevice.fbPower;
      _stMsg.iErrorNumber           := 0;

      _stMsg.sText                  := concat('clear error on disable : ', TO_STRING(_eResult));

      IF (_MessageLevel = E_MessageType.eMessageVerbose)
      THEN
        f_MessageSet(_stMsg);
      END_IF
    END_IF
END_CASE
CASE _eState
OF
  E_PROGRESS.PROGRESS_OCCUPIED:
    IF _AxisRef.Status.Error
    THEN
      _nErrorId                     := _AxisRef.NcToPlc.ErrorCode;
    
      _stMsg.eType                  := E_MessageType.eMessageError;
      _stMsg.eDevice                := e_Device.Axis + (_AxisRef.NcToPlc.AxisId);
      _stMsg.eSubdevice             :=  e_SubDevice.fbPower;
      _stMsg.iErrorNumber           := _nErrorId;

      f_MessageSet(_stMsg);
    
      _eState                       := E_PROGRESS.PROGRESS_ERROR;

    ELSIF NOT _AxisRef.Status.ControlLoopClosed
    THEN
      _eState                       := E_PROGRESS.PROGRESS_WORKING;
    END_IF
END_CASE
CASE _eState
OF
  E_PROGRESS.PROGRESS_WORKING:
    _eResult                        := Reset(FALSE);
    _eState                         := E_PROGRESS.PROGRESS_DONE;

      _stMsg.eType                  := E_MessageType.eMessageVerbose;
      _stMsg.eDevice                := E_Device.Axis + (_AxisRef.NcToPlc.AxisId);
      _stMsg.eSubdevice             := e_Subdevice.fbPower;
      _stMsg.iErrorNumber           := 0;

      _stMsg.sText                  := concat(' : ', TO_STRING(_eState));

      IF (_MessageLevel = E_MessageType.eMessageVerbose)
      THEN
        f_MessageSet(_stMsg);
      END_IF
END_CASE

Disable                             := _eState;
END_METHOD

METHOD Enable : E_PROGRESS
VAR_INPUT
  Execute           : BOOL;
END_VAR
VAR_INST
  _eResult,
  _eState           : E_PROGRESS;
  _rValue           : LREAL;
  _stMsg            : ST_Message;
END_VAR
IF NOT (__ISVALIDREF(_AxisRef)) THEN  Enable  := E_PROGRESS.PROGRESS_ERROR; RETURN; END_IF
IF NOT Execute THEN _eState := E_PROGRESS.PROGRESS_INIT; END_IF

CASE _eState
OF
  E_PROGRESS.PROGRESS_INIT:
    IF Execute 
    THEN
      memset(ADR(_stMsg),0,SIZEOF(_stMsg));
      _nErrorId                     := 0;
      _rValue                       := 0;
      _eState                       := E_PROGRESS.PROGRESS_BUSY;
    END_IF
END_CASE
CASE _eState
OF
  E_PROGRESS.PROGRESS_BUSY:
    _fbPower.Enable                 := TRUE;
    _eResult                        := Reset(FALSE);
    _eState                         := E_PROGRESS.PROGRESS_STARTUP;

  E_PROGRESS.PROGRESS_STARTUP:
    IF _fbPower.Error OR
       _AxisRef.Status.Error
    THEN
      _eState                       := E_PROGRESS.PROGRESS_PREPARE;

      _stMsg.eType                  := E_MessageType.eMessageVerbose;
      _stMsg.eDevice                := E_Device.Axis + (_AxisRef.NcToPlc.AxisId);
      _stMsg.eSubdevice             := e_Subdevice.fbPower;
      _stMsg.iErrorNumber           := 0;

      _stMsg.sText                  := concat('clear error on enable : ', TO_STRING(_eState));

      IF (_MessageLevel = E_MessageType.eMessageVerbose)
      THEN
        f_MessageSet(_stMsg);
      END_IF
    ELSE
      _eState                       := E_PROGRESS.PROGRESS_OCCUPIED;
    END_IF
END_CASE
CASE _eState
OF
  E_PROGRESS.PROGRESS_PREPARE:
    _eResult                        := Reset(TRUE);
    IF (_eResult = E_PROGRESS.PROGRESS_DONE)
    THEN
      _eState                       := E_PROGRESS.PROGRESS_OCCUPIED;
    END_IF
END_CASE
CASE _eState
OF
  E_PROGRESS.PROGRESS_OCCUPIED:
    IF _AxisRef.Status.Error
    THEN
      _nErrorId                     := _AxisRef.NcToPlc.ErrorCode;
    
      _stMsg.eType                  := E_MessageType.eMessageError;
      _stMsg.eDevice                := e_Device.Axis + (_AxisRef.NcToPlc.AxisId);
      _stMsg.eSubdevice             :=  e_SubDevice.fbPower;
      _stMsg.iErrorNumber           := _nErrorId;
    
      f_MessageSet(_stMsg);

      _eState                       := E_PROGRESS.PROGRESS_ERROR;

    ELSIF _AxisRef.Status.ControlLoopClosed
    THEN
      _eState                       := E_PROGRESS.PROGRESS_WORKING;
    END_IF
END_CASE
CASE _eState
OF
  E_PROGRESS.PROGRESS_WORKING:
    _eResult                        := Reset(FALSE);
    _eState                         := E_PROGRESS.PROGRESS_DONE;

      _stMsg.eType                  := E_MessageType.eMessageVerbose;
      _stMsg.eDevice                := E_Device.Axis + (_AxisRef.NcToPlc.AxisId);
      _stMsg.eSubdevice             := e_Subdevice.fbPower;
      _stMsg.iErrorNumber           := 0;

      _stMsg.sText                  := concat(' : ', TO_STRING(_eState));

      IF (_MessageLevel = E_MessageType.eMessageVerbose)
      THEN
        f_MessageSet(_stMsg);
      END_IF
END_CASE

Enable                              := _eState;
END_METHOD

PROPERTY EncoderType : E_AxisEncoderType
GET
EncoderType := _eEncoderType;
END_GET
END_PROPERTY

PROPERTY ErrorId : udint
GET
ErrorId := _nErrorId;
END_GET
END_PROPERTY

METHOD Halt : E_PROGRESS
VAR_INPUT
  Execute           : BOOL;
  Dec               : LREAL;
  Jerk              : LREAL;
END_VAR
VAR_INST
  _eState           : E_PROGRESS;
  _rValue           : LREAL;
  _stMsg            : ST_Message;
END_VAR
IF NOT (__ISVALIDREF(_AxisRef)) THEN  Halt  := E_PROGRESS.PROGRESS_ERROR; RETURN; END_IF
IF NOT Execute THEN _eState := E_PROGRESS.PROGRESS_INIT; END_IF

CASE _eState
OF
  E_PROGRESS.PROGRESS_INIT:
    IF Execute 
    THEN
      memset(ADR(_stMsg),0,SIZEOF(_stMsg));
      _nErrorId                     := 0;
      _rValue                       := 0;
      _eState                       := E_PROGRESS.PROGRESS_BUSY;
    END_IF
END_CASE
CASE _eState
OF
  E_PROGRESS.PROGRESS_BUSY:
    _eState                         := E_PROGRESS.PROGRESS_OCCUPIED;
    _fbHalt(
              Axis                  := _AxisRef, 
              Execute               := FALSE, 
              Deceleration          := Dec, 
              Jerk                  := Jerk, 
              BufferMode            := Tc2_MC2.MC_BufferMode.MC_Aborting);
END_CASE
CASE _eState
OF
  E_PROGRESS.PROGRESS_OCCUPIED:
    _fbHalt(
              Axis                  := _AxisRef, 
              Execute               := TRUE, 
              Deceleration          := Dec, 
              Jerk                  := Jerk, 
              BufferMode            := Tc2_MC2.MC_BufferMode.MC_Aborting);

    IF _fbhalt.Error
    THEN
      _eState                       := E_PROGRESS.PROGRESS_ERROR;
        _nErrorId                   := _fbHalt.ErrorID;

        _stMsg.eType                := E_MessageType.eMessageError;
        _stMsg.eDevice              := e_Device.Axis + (_AxisRef.NcToPlc.AxisId);
        _stMsg.eSubdevice           := e_SubDevice.fbHalt;
        _stMsg.iErrorNumber         := _nErrorId;

        _stMsg.sText                := concat(' : ', TO_STRING(_eState));

        f_MessageSet(_stMsg);

        _fbHalt(
              Axis                  := _AxisRef, 
              Execute               := FALSE);
    ELSE
      IF _fbHalt.Done OR
         _AxisRef.Status.NotMoving
      THEN
        _eState                     := E_PROGRESS.PROGRESS_WORKING;

      ELSIF _fbHalt.CommandAborted
      THEN
        _eState                     := E_PROGRESS.PROGRESS_BUSY;

        _stMsg.eType                := E_MessageType.eMessageWarning;
        _stMsg.eDevice              := E_Device.Axis + (_AxisRef.NcToPlc.AxisId);
        _stMsg.eSubdevice           := e_Subdevice.fbHalt;
        _stMsg.iErrorNumber         := 0;
    
        _stMsg.sText                := concat('command aborted : ', TO_STRING(_eState));

        IF (_MessageLevel > E_MessageType.eMessageError)
        THEN
          f_MessageSet(_stMsg);
        END_IF
      END_IF
    END_IF
END_CASE
CASE _eState
OF
  E_PROGRESS.PROGRESS_WORKING:
    _fbHalt(
              Axis                  := _AxisRef, 
              Execute               := FALSE);

    _eState                         := E_PROGRESS.PROGRESS_DONE;

    _stMsg.eType                    := E_MessageType.eMessageVerbose;
    _stMsg.eDevice                  := E_Device.Axis + (_AxisRef.NcToPlc.AxisId);
    _stMsg.eSubdevice               := e_Subdevice.fbHalt;
    _stMsg.iErrorNumber             := 0;

    _stMsg.sText                    := concat(' : ', TO_STRING(_eState));

    IF (_MessageLevel = E_MessageType.eMessageVerbose)
    THEN
      f_MessageSet(_stMsg);
    END_IF
END_CASE

Halt := _eState;
END_METHOD

METHOD Home : E_PROGRESS
VAR_INPUT
  Execute           : BOOL;
  Position          : LREAL := DEFAULT_HOME_POSITION;
  HomingMode        : Tc2_MC2.MC_HomingMode := MC_DefaultHoming;
  Options           : Tc2_MC2.ST_HomingOptions;
END_VAR
VAR_INST
  _eState           : E_PROGRESS;
  _sValue           : STRING(40);
  _rValue           : LREAL;
  _stMsg            : ST_Message;
END_VAR
IF NOT (__ISVALIDREF(_AxisRef)) THEN  Home  := E_PROGRESS.PROGRESS_ERROR; RETURN; END_IF
IF NOT Execute THEN _eState := E_PROGRESS.PROGRESS_INIT; END_IF

CASE _eState
OF
  E_PROGRESS.PROGRESS_INIT:
    IF Execute 
    THEN
      memset(ADR(_stMsg), 0,SIZEOF(_stMsg));
      memset(ADR(_sValue),0,SIZEOF(_sValue));

      _nErrorId                     := 0;
      _rValue                       := 0;
      _eState                       := E_PROGRESS.PROGRESS_BUSY;

      IF NOT (_pCalibrationCam <> 0) 
      THEN
        _eState                     := E_PROGRESS.PROGRESS_ERROR;
        // prevent page fault
        _sValue                     := 'Pointer to calibration cam not set';

        _nErrorId                   := 666;

        _stMsg.eType                := E_MessageType.eMessageError;
        _stMsg.eDevice              := e_Device.Axis + (_AxisRef.NcToPlc.AxisId);
        _stMsg.eSubdevice           := e_SubDevice.fbHome;
        _stMsg.iErrorNumber         := _nErrorId;
        _stMsg.sText                := _sValue;

        f_MessageSet(_stMsg);
      END_IF
    END_IF
END_CASE
CASE _eState
OF
  E_PROGRESS.PROGRESS_BUSY:
    _eState                         := E_PROGRESS.PROGRESS_OCCUPIED;
    _fbHome(
            Axis                    := _AxisRef, 
            Execute                 := FALSE, 
            Position                := Position, 
            HomingMode              := HomingMode, 
            Options                 := Options, 
            bCalibrationCam         := _pCalibrationCam^);
END_CASE
CASE _eState
OF
  E_PROGRESS.PROGRESS_OCCUPIED:
    _fbHome(
            Execute                 := TRUE, 
            Axis                    := _AxisRef);

    IF _fbHome.Done
    THEN
      _eState                       := E_PROGRESS.PROGRESS_WORKING;
    ELSE
      IF _fbHome.Error
      THEN
        _eState                     := E_PROGRESS.PROGRESS_ERROR;
        _nErrorId                   := _fbHome.ErrorID;

        _stMsg.eType                := E_MessageType.eMessageError;
        _stMsg.eDevice              := e_Device.Axis + (_AxisRef.NcToPlc.AxisId);
        _stMsg.eSubdevice           :=  e_SubDevice.fbHome;
        _stMsg.iErrorNumber         := _nErrorId;

        f_MessageSet(_stMsg);

        _fbHome(
            Execute                 := FALSE, 
            Axis                    := _AxisRef);
      END_IF
    END_IF
END_CASE
CASE _eState
OF
  E_PROGRESS.PROGRESS_WORKING:
    _fbHome(
            Execute                 := FALSE, 
            Axis                    := _AxisRef);

    _eState                         := E_PROGRESS.PROGRESS_DONE;

    _stMsg.eType                    := E_MessageType.eMessageVerbose;
    _stMsg.eDevice                  := E_Device.Axis + (_AxisRef.NcToPlc.AxisId);
    _stMsg.eSubdevice               := e_Subdevice.fbHome;
    _stMsg.iErrorNumber             := 0;

    _stMsg.sText                    := concat(' : ', TO_STRING(_eState));
    IF (_MessageLevel = E_MessageType.eMessageVerbose)
    THEN
      f_MessageSet(_stMsg);
    END_IF
END_CASE

Home                                := _eState;
END_METHOD

PROPERTY LastTargetPosition : LREAL
GET
END_GET
END_PROPERTY

PROPERTY MessageLevel : E_MessageType
SET
_MessageLevel := MessageLevel;
END_SET
END_PROPERTY

METHOD MovePosBuffer : E_PROGRESS
VAR_INPUT
  bEnable          : BOOL;
  Position        : LREAL;
  Vel             : LREAL;
  Acc             : LREAL;
  Dec             : LREAL;
  Jerk            : LREAL;
  BufferMode      : Tc2_MC2.MC_BufferMode;
END_VAR
VAR_INST
  _eState           : E_PROGRESS;
  _rValue           : LREAL;
  _stMsg            : ST_Message;
END_VAR
IF NOT (__ISVALIDREF(_AxisRef)) THEN  MovePosBuffer  := E_PROGRESS.PROGRESS_ERROR; RETURN; END_IF
IF NOT bEnable THEN _eState := E_PROGRESS.PROGRESS_INIT; END_IF

CASE _eState
OF
  E_PROGRESS.PROGRESS_INIT:
    IF bEnable 
    THEN
      memset(ADR(_stMsg),0,SIZEOF(_stMsg));
      _nErrorId                     := 0;
      _rValue                       := Position;

      _eState                       := E_PROGRESS.PROGRESS_BUSY;

      _stMsg.eType                  := E_MessageType.eMessageVerbose;
      _stMsg.eDevice                := e_Device.Axis + (_AxisRef.NcToPlc.AxisId);
      _stMsg.eSubdevice             := e_SubDevice.fbMoveAbsolute1;
      _stMsg.iErrorNumber           := 0;

      _stMsg.sText                  := concat('FB start : ', TO_STRING(_rValue));

      IF (_MessageLevel = E_MessageType.eMessageVerbose)
      THEN
        f_MessageSet(_stMsg);
      END_IF
    END_IF
END_CASE
CASE _eState
OF
  E_PROGRESS.PROGRESS_BUSY:
    _eState                         := E_PROGRESS.PROGRESS_STARTUP;
    _fbMoveAbsolute[1](
                    Axis            := _AxisRef,
                    Execute         := FALSE);

    _fbMoveAbsolute[2](
                    Axis            := _AxisRef,
                    Execute         := FALSE);

END_CASE
CASE _eState
OF
  E_PROGRESS.PROGRESS_STARTUP:
    _fbMoveAbsolute[1](
                    Axis            := _AxisRef, 
                    Execute         := TRUE,
                    Position        := _rValue, 
                    Velocity        := Vel, 
                    Acceleration    := Acc, 
                    Deceleration    := Dec, 
                    Jerk            := Jerk, 
                    BufferMode      := BufferMode);

    _fbMoveAbsolute[2](
                    Axis            := _AxisRef,
                    Execute         := FALSE);

    _rLastTargetPosition            := _fbMoveAbsolute[1].Position;

    IF _fbMoveAbsolute[1].Error
    THEN
      _eState                       := E_PROGRESS.PROGRESS_ERROR;
      _nErrorId                     := _fbMoveAbsolute[1].ErrorID;
    
      _stMsg.eType                  := E_MessageType.eMessageError;
      _stMsg.eDevice                := e_Device.Axis + (_AxisRef.NcToPlc.AxisId);
      _stMsg.eSubdevice             :=  e_SubDevice.fbMoveAbsolute1;
      _stMsg.iErrorNumber           := _nErrorId;
    
      _stMsg.sText                  := concat(' : ', TO_STRING(_eState));
    
      f_MessageSet(_stMsg);

    ELSIF (_fbMoveAbsolute[1].Busy)
    THEN
      _eState                       := E_PROGRESS.PROGRESS_PREPARE;

      _stMsg.eType                  := E_MessageType.eMessageVerbose;
      _stMsg.eDevice                := e_Device.Axis + (_AxisRef.NcToPlc.AxisId);
      _stMsg.eSubdevice             :=  e_SubDevice.fbMoveAbsolute1;
      _stMsg.iErrorNumber           := 0;

      _stMsg.sText                  := concat('FB busy: ', TO_STRING(_eState));

      IF (_MessageLevel = E_MessageType.eMessageVerbose)
      THEN
        f_MessageSet(_stMsg);
      END_IF

    ELSIF (_fbMoveAbsolute[1].CommandAborted)
    THEN
      _eState                       := E_PROGRESS.PROGRESS_PREPARE;

      _stMsg.eType                  := E_MessageType.eMessageVerbose;
      _stMsg.eDevice                := e_Device.Axis + (_AxisRef.NcToPlc.AxisId);
      _stMsg.eSubdevice             :=  e_SubDevice.fbMoveAbsolute1;
      _stMsg.iErrorNumber           := 0;

      _stMsg.sText                  := concat('FB aborted: ', TO_STRING(_eState));

      IF (_MessageLevel = E_MessageType.eMessageVerbose)
      THEN
        f_MessageSet(_stMsg);
      END_IF

    ELSIF (_fbMoveAbsolute[1].Done)
    THEN
      _eState                       := E_PROGRESS.PROGRESS_PREPARE;

      _stMsg.eType                  := E_MessageType.eMessageVerbose;
      _stMsg.eDevice                := e_Device.Axis + (_AxisRef.NcToPlc.AxisId);
      _stMsg.eSubdevice             :=  e_SubDevice.fbMoveAbsolute1;
      _stMsg.iErrorNumber           := 0;

      _stMsg.sText                  := concat('FB done: ', TO_STRING(_eState));

      IF (_MessageLevel = E_MessageType.eMessageVerbose)
      THEN
        f_MessageSet(_stMsg);
      END_IF
    END_IF
END_CASE
CASE _eState
OF
  E_PROGRESS.PROGRESS_PREPARE:
    _fbMoveAbsolute[1](
                    Axis            := _AxisRef);
    _fbMoveAbsolute[2](
                    Axis            := _AxisRef,
                    Execute         := FALSE);

    IF _fbMoveAbsolute[1].Error
    THEN
      _eState                       := E_PROGRESS.PROGRESS_ERROR;
      _nErrorId                     := _fbMoveAbsolute[1].ErrorID;
    
      _stMsg.eType                  := E_MessageType.eMessageError;
      _stMsg.eDevice                := e_Device.Axis + (_AxisRef.NcToPlc.AxisId);
      _stMsg.eSubdevice             :=  e_SubDevice.fbMoveAbsolute1;
      _stMsg.iErrorNumber           := _nErrorId;
    
      _stMsg.sText                  := concat(' : ', TO_STRING(_eState));
    
      f_MessageSet(_stMsg);

    ELSIF (Position <> _rValue)
    THEN
      IF _fbMoveAbsolute[1].Active
      THEN
        _fbMoveAbsolute[1](
                    Axis            := _AxisRef, 
                    Execute         := FALSE);
  
        _eState                       := E_PROGRESS.PROGRESS_CHECK;
  
        _stMsg.eType                  := E_MessageType.eMessageVerbose;
        _stMsg.eDevice                := e_Device.Axis + (_AxisRef.NcToPlc.AxisId);
        _stMsg.eSubdevice             :=  e_SubDevice.fbMoveAbsolute2;
        _stMsg.iErrorNumber           := 0;
  
        _stMsg.sText                  := concat('Position changed: ', TO_STRING(_rValue));
        _stMsg.sText                  := concat(_stMsg.sText        , ' to ');
        _stMsg.sText                  := concat(_stMsg.sText        , TO_STRING(Position));
  
        IF (_MessageLevel = E_MessageType.eMessageVerbose)
        THEN
          f_MessageSet(_stMsg);
        END_IF

        _rValue                       := Position;
      END_IF
    END_IF
END_CASE
CASE _eState
OF
  E_PROGRESS.PROGRESS_CHECK:
    _fbMoveAbsolute[1](
                    Axis            := _AxisRef,
                    Execute         := FALSE);

    _fbMoveAbsolute[2](
                    Axis            := _AxisRef, 
                    Execute         := TRUE,
                    Position        := _rValue, 
                    Velocity        := Vel, 
                    Acceleration    := Acc, 
                    Deceleration    := Dec, 
                    Jerk            := Jerk, 
                    BufferMode      := BufferMode);

    _rLastTargetPosition            := _fbMoveAbsolute[2].Position;

    IF _fbMoveAbsolute[2].Error
    THEN
      _eState                       := E_PROGRESS.PROGRESS_ERROR;
      _nErrorId                     := _fbMoveAbsolute[2].ErrorID;
    
      _stMsg.eType                  := E_MessageType.eMessageError;
      _stMsg.eDevice                := e_Device.Axis + (_AxisRef.NcToPlc.AxisId);
      _stMsg.eSubdevice             :=  e_SubDevice.fbMoveAbsolute2;
      _stMsg.iErrorNumber           := _nErrorId;
    
      _stMsg.sText                  := concat(' : ', TO_STRING(_eState));
    
      f_MessageSet(_stMsg);

    ELSIF (_fbMoveAbsolute[2].Busy)
    THEN
      _eState                       := E_PROGRESS.PROGRESS_OCCUPIED;

      _stMsg.eType                  := E_MessageType.eMessageVerbose;
      _stMsg.eDevice                := e_Device.Axis + (_AxisRef.NcToPlc.AxisId);
      _stMsg.eSubdevice             :=  e_SubDevice.fbMoveAbsolute2;
      _stMsg.iErrorNumber           := 0;

      _stMsg.sText                  := concat('FB busy: ', TO_STRING(_eState));

      IF (_MessageLevel = E_MessageType.eMessageVerbose)
      THEN
        f_MessageSet(_stMsg);
      END_IF

    ELSIF (_fbMoveAbsolute[2].CommandAborted)
    THEN
      _eState                       := E_PROGRESS.PROGRESS_OCCUPIED;

      _stMsg.eType                  := E_MessageType.eMessageVerbose;
      _stMsg.eDevice                := e_Device.Axis + (_AxisRef.NcToPlc.AxisId);
      _stMsg.eSubdevice             :=  e_SubDevice.fbMoveAbsolute2;
      _stMsg.iErrorNumber           := 0;

      _stMsg.sText                  := concat('FB aborted: ', TO_STRING(_eState));

      IF (_MessageLevel = E_MessageType.eMessageVerbose)
      THEN
        f_MessageSet(_stMsg);
      END_IF

    ELSIF (_fbMoveAbsolute[2].Done)
    THEN
      _eState                       := E_PROGRESS.PROGRESS_OCCUPIED;

      _stMsg.eType                  := E_MessageType.eMessageVerbose;
      _stMsg.eDevice                := e_Device.Axis + (_AxisRef.NcToPlc.AxisId);
      _stMsg.eSubdevice             :=  e_SubDevice.fbMoveAbsolute2;
      _stMsg.iErrorNumber           := 0;

      _stMsg.sText                  := concat('FB done: ', TO_STRING(_eState));

      IF (_MessageLevel = E_MessageType.eMessageVerbose)
      THEN
        f_MessageSet(_stMsg);
      END_IF
    END_IF
END_CASE
CASE _eState
OF
  E_PROGRESS.PROGRESS_OCCUPIED:
    _fbMoveAbsolute[1](
                    Axis            := _AxisRef,
                    Execute         := FALSE);

    _fbMoveAbsolute[2](
                    Axis            := _AxisRef);

    IF _fbMoveAbsolute[2].Error
    THEN
      _eState                       := E_PROGRESS.PROGRESS_ERROR;
      _nErrorId                     := _fbMoveAbsolute[2].ErrorID;
    
      _stMsg.eType                  := E_MessageType.eMessageError;
      _stMsg.eDevice                := e_Device.Axis + (_AxisRef.NcToPlc.AxisId);
      _stMsg.eSubdevice             :=  e_SubDevice.fbMoveAbsolute2;
      _stMsg.iErrorNumber           := _nErrorId;
    
      _stMsg.sText                  := concat(' : ', TO_STRING(_eState));
    
      f_MessageSet(_stMsg);

    ELSIF (Position <> _rValue)
    THEN
      IF _fbMoveAbsolute[2].Active
      THEN
        _fbMoveAbsolute[2](Axis       := _AxisRef,
                           Execute    := FALSE);
  
        _eState                       := E_PROGRESS.PROGRESS_STARTUP;
  
        _stMsg.eType                  := E_MessageType.eMessageVerbose;
        _stMsg.eDevice                := e_Device.Axis + (_AxisRef.NcToPlc.AxisId);
        _stMsg.eSubdevice             :=  e_SubDevice.fbMoveAbsolute1;
        _stMsg.iErrorNumber           := 0;
  
        _stMsg.sText                  := concat('Position changed: ', TO_STRING(_rValue));
        _stMsg.sText                  := concat(_stMsg.sText        , ' to ');
        _stMsg.sText                  := concat(_stMsg.sText        , TO_STRING(Position));
  
        IF (_MessageLevel = E_MessageType.eMessageVerbose)
        THEN
          f_MessageSet(_stMsg);
        END_IF
 
        _rValue                       := Position;
      END_IF
    END_IF
END_CASE
CASE _eState
OF
  E_PROGRESS.PROGRESS_INIT,
  E_PROGRESS.PROGRESS_ERROR:
    _fbMoveAbsolute[1](
                    Axis            := _AxisRef,
                    Execute         := FALSE);

    _fbMoveAbsolute[2](
                    Axis            := _AxisRef,
                    Execute         := FALSE);
END_CASE


MovePosBuffer                       := _eState;
END_METHOD

METHOD MoveToPos : E_PROGRESS
VAR_INPUT
  Execute         : BOOL;
  Position        : LREAL;
  Vel             : LREAL;
  Acc             : LREAL;
  Dec             : LREAL;
  Jerk            : LREAL;
  BufferMode      : Tc2_MC2.MC_BufferMode;
END_VAR
VAR_INST
  _eState           : E_PROGRESS;
  _rValue           : LREAL;
  _stMsg            : ST_Message;
END_VAR
IF NOT (__ISVALIDREF(_AxisRef)) THEN  MoveToPos  := E_PROGRESS.PROGRESS_ERROR; RETURN; END_IF
IF NOT Execute THEN _eState := E_PROGRESS.PROGRESS_INIT; END_IF

CASE _eState
OF
  E_PROGRESS.PROGRESS_INIT:
    IF Execute 
    THEN
      memset(ADR(_stMsg),0,SIZEOF(_stMsg));
      _nErrorId                     := 0;
      _rValue                       := 0;
      _eState                       := E_PROGRESS.PROGRESS_BUSY;

      _stMsg.eType                  := E_MessageType.eMessageInfo;
      _stMsg.eDevice                := e_Device.Axis + (_AxisRef.NcToPlc.AxisId);
      _stMsg.eSubdevice             := e_SubDevice.fbMovePtP;
      _stMsg.iErrorNumber           := 0;

      _stMsg.sText                  := concat(' : ', TO_STRING(Position));

      IF (_MessageLevel > E_MessageType.eMessageError)
      THEN
        f_MessageSet(_stMsg);
      END_IF
    END_IF
END_CASE
CASE _eState
OF
  E_PROGRESS.PROGRESS_BUSY:
    _eState                         := E_PROGRESS.PROGRESS_STARTUP;
    _rValue                         := Position;

    _fbMoveToPosition(
                    Axis            := _AxisRef,
                    Execute         := FALSE);
END_CASE
CASE _eState
OF
  E_PROGRESS.PROGRESS_STARTUP:
    _eState                         := E_PROGRESS.PROGRESS_PREPARE;
    _fbMoveToPosition(
                    Axis            := _AxisRef, 
                    Execute         := TRUE,
                    Position        := _rValue, 
                    Velocity        := Vel, 
                    Acceleration    := Acc, 
                    Deceleration    := Dec, 
                    Jerk            := Jerk, 
                    BufferMode      := BufferMode);

    _rLastTargetPosition            := _fbMoveToPosition.Position;
END_CASE
CASE _eState
OF
  E_PROGRESS.PROGRESS_PREPARE:
    _fbMoveToPosition(
                    Axis            := _AxisRef);

    IF (_fbMoveToPosition.Error)
    THEN
      _eState                       := E_PROGRESS.PROGRESS_ERROR;
      _nErrorId                     := _fbMoveToPosition.ErrorID;
    
      _stMsg.eType                  := E_MessageType.eMessageError;
      _stMsg.eDevice                := e_Device.Axis + (_AxisRef.NcToPlc.AxisId);
      _stMsg.eSubdevice             :=  e_SubDevice.fbMovePtP;
      _stMsg.iErrorNumber           := _nErrorId;

      _stMsg.sText                  := concat(' : ', TO_STRING(_eState));
    
      f_MessageSet(_stMsg);

    ELSIF (_fbMoveToPosition.CommandAborted)
    THEN
      _eState                       := E_PROGRESS.PROGRESS_ERROR;
      _nErrorId                     := _fbMoveToPosition.ErrorID;

      _stMsg.eType                  := E_MessageType.eMessageError;
      _stMsg.eDevice                := e_Device.Axis + (_AxisRef.NcToPlc.AxisId);
      _stMsg.eSubdevice             := e_SubDevice.fbMovePtP;
      _stMsg.iErrorNumber           := _nErrorId;

      _stMsg.sText                  := concat('FB aborted: ', TO_STRING(_eState));

      f_MessageSet(_stMsg);

    ELSIF (_fbMoveToPosition.Active)
    THEN
      _eState                       := E_PROGRESS.PROGRESS_OCCUPIED;

      _stMsg.eType                  := E_MessageType.eMessageVerbose;
      _stMsg.eDevice                := e_Device.Axis + (_AxisRef.NcToPlc.AxisId);
      _stMsg.eSubdevice             := e_SubDevice.fbMovePtP;
      _stMsg.iErrorNumber           := 0;

      _stMsg.sText                  := concat('FB active: ', TO_STRING(_eState));

      IF (_MessageLevel = E_MessageType.eMessageVerbose)
      THEN
        f_MessageSet(_stMsg);
      END_IF

    ELSIF (_fbMoveToPosition.Done)
    THEN
      _eState                       := E_PROGRESS.PROGRESS_STILL_WORKING;
    END_IF
END_CASE
CASE _eState
OF
  E_PROGRESS.PROGRESS_OCCUPIED:
    _fbMoveToPosition(
                    Axis            := _AxisRef);

    IF (_fbMoveToPosition.Error)
    THEN
      _eState                       := E_PROGRESS.PROGRESS_ERROR;
      _nErrorId                     := _fbMoveToPosition.ErrorID;
    
      _stMsg.eType                  := E_MessageType.eMessageError;
      _stMsg.eDevice                := e_Device.Axis + (_AxisRef.NcToPlc.AxisId);
      _stMsg.eSubdevice             :=  e_SubDevice.fbMovePtP;
      _stMsg.iErrorNumber           := _nErrorId;

      _stMsg.sText                  := concat(' : ', TO_STRING(_eState));

      f_MessageSet(_stMsg);

    ELSIF (_fbMoveToPosition.CommandAborted)
    THEN
      _eState                       := E_PROGRESS.PROGRESS_ERROR;
      _nErrorId                     := _fbMoveToPosition.ErrorID;
    
      _stMsg.eType                  := E_MessageType.eMessageError;
      _stMsg.eDevice                := e_Device.Axis + (_AxisRef.NcToPlc.AxisId);
      _stMsg.eSubdevice             :=  e_SubDevice.fbMovePtP;
      _stMsg.iErrorNumber           := _nErrorId;

      _stMsg.sText                  := concat('FB aborted : ', TO_STRING(_eState));

      f_MessageSet(_stMsg);

    ELSIF (_fbMoveToPosition.Done)
    THEN
      _eState                       := E_PROGRESS.PROGRESS_STILL_WORKING;
    END_IF
END_CASE
CASE _eState
OF
  E_PROGRESS.PROGRESS_STILL_WORKING:
    _eState                         := E_PROGRESS.PROGRESS_DONE;

    _fbMoveToPosition(
                  Axis              := _AxisRef,
                  Execute           := FALSE);

    _stMsg.eType                    := E_MessageType.eMessageVerbose;
    _stMsg.eDevice                  := e_Device.Axis + (_AxisRef.NcToPlc.AxisId);
    _stMsg.eSubdevice               := e_SubDevice.fbMovePtP;
    _stMsg.iErrorNumber             := 0;

    _stMsg.sText                    := concat(' : ', TO_STRING(_eState));

    IF (_MessageLevel = E_MessageType.eMessageVerbose)
    THEN
      f_MessageSet(_stMsg);
    END_IF
END_CASE

MoveToPos                           := _eState;
END_METHOD

METHOD MoveVelo : E_PROGRESS
VAR_INPUT
  Execute           : BOOL;
  Velocity          : LREAL;
  Acc               : LREAL;
  Dec               : LREAL;
  Jerk              : LREAL;
  Direction         : Tc2_MC2.MC_Direction := MC_Positive_Direction;
  BufferMode        : Tc2_MC2.MC_BufferMode;
END_VAR
VAR_INST
  _eState           : E_PROGRESS;
  _rValue           : LREAL;
  _stMsg            : ST_Message;
END_VAR
IF NOT (__ISVALIDREF(_AxisRef)) THEN  MoveVelo  := E_PROGRESS.PROGRESS_ERROR; RETURN; END_IF
IF NOT Execute THEN _eState := E_PROGRESS.PROGRESS_INIT; END_IF

CASE _eState
OF
  E_PROGRESS.PROGRESS_INIT:
    IF Execute 
    THEN
      memset(ADR(_stMsg),0,SIZEOF(_stMsg));
      _nErrorId                     := 0;
      _rValue                       := Velocity;
      _eState                       := E_PROGRESS.PROGRESS_BUSY;

      _stMsg.eType                  := E_MessageType.eMessageInfo;
      _stMsg.eDevice                := e_Device.Axis + (_AxisRef.NcToPlc.AxisId);
      _stMsg.eSubdevice             := e_SubDevice.fbMoveVelo;
      _stMsg.iErrorNumber           := 0;

      _stMsg.sText                  := concat('FB start : ', TO_STRING(_rValue));

      IF (_MessageLevel > E_MessageType.eMessageError)
      THEN
        f_MessageSet(_stMsg);
      END_IF
    END_IF
END_CASE
CASE _eState
OF
  E_PROGRESS.PROGRESS_BUSY:
    _eState                         := E_PROGRESS.PROGRESS_STARTUP;
    _fbMoveVelo(
                      Axis          := _AxisRef, 
                      Execute       := FALSE, 
                      Velocity      := _rValue, 
                      Acceleration  := Acc, 
                      Deceleration  := Dec, 
                      Jerk          := Jerk, 
                      Direction     := Direction, 
                      BufferMode    := BufferMode);
END_CASE
CASE _eState
OF
  E_PROGRESS.PROGRESS_STARTUP:
    _fbMoveVelo(
                      Axis          := _AxisRef, 
                      Execute       := TRUE);
    _eState                         := E_PROGRESS.PROGRESS_OCCUPIED;
END_CASE
CASE _eState
OF
  E_PROGRESS.PROGRESS_OCCUPIED:
    _fbMoveVelo(
                      Axis          := _AxisRef);

    IF _fbMoveVelo.Error
    THEN
      _eState                       := E_PROGRESS.PROGRESS_ERROR;
      _nErrorId                     := _fbMoveVelo.ErrorID;
    
      _stMsg.eType                  := E_MessageType.eMessageError;
      _stMsg.eDevice                := e_Device.Axis + (_AxisRef.NcToPlc.AxisId);
      _stMsg.eSubdevice             :=  e_SubDevice.fbMoveVelo;
      _stMsg.iErrorNumber           := _nErrorId;

      _stMsg.sText                  := concat(' : ', TO_STRING(_eState));

      f_MessageSet(_stMsg);

      _fbMoveVelo(
                      Axis          := _AxisRef, 
                      Execute       := FALSE);

    ELSIF _fbMoveVelo.CommandAborted
    THEN
      _eState                       := E_PROGRESS.PROGRESS_ERROR;

      _nErrorId                     := _fbMoveVelo.ErrorID;
    
      _stMsg.eType                  := E_MessageType.eMessageError;
      _stMsg.eDevice                := e_Device.Axis + (_AxisRef.NcToPlc.AxisId);
      _stMsg.eSubdevice             :=  e_SubDevice.fbMoveVelo;
      _stMsg.iErrorNumber           := _nErrorId;

      _stMsg.sText                  := concat('FB aborted : ', TO_STRING(_eState));

      f_MessageSet(_stMsg);

      _fbMoveVelo(
                      Axis          := _AxisRef, 
                      Execute       := FALSE);
    
    ELSIF _fbMoveVelo.InVelocity
    THEN
      _eState                       := E_PROGRESS.PROGRESS_WORKING;
    END_IF
END_CASE
CASE _eState
OF
  E_PROGRESS.PROGRESS_WORKING:
    _fbMoveVelo(
                      Axis          := _AxisRef, 
                      Execute       := FALSE);

    _eState                         := E_PROGRESS.PROGRESS_DONE;

    _stMsg.eType                    := E_MessageType.eMessageVerbose;
    _stMsg.eDevice                  := e_Device.Axis + (_AxisRef.NcToPlc.AxisId);
    _stMsg.eSubdevice               := e_SubDevice.fbMoveVelo;
    _stMsg.iErrorNumber             := 0;

    _stMsg.sText                    := concat('FB InVelocity : ', TO_STRING(_eState));

    IF (_MessageLevel = E_MessageType.eMessageVerbose)
    THEN
      f_MessageSet(_stMsg);
    END_IF
END_CASE


MoveVelo                            := _eState;
END_METHOD

METHOD MoveVeloBuffer : E_PROGRESS
VAR_INPUT
  bEnable          : BOOL;
  Velocity        : LREAL;
  Acc             : LREAL;
  Dec             : LREAL;
  Jerk            : LREAL;
  BufferMode      : Tc2_MC2.MC_BufferMode;
END_VAR
VAR_INST
  _eState           : E_PROGRESS;
  _rValue           : LREAL;
  _stMsg            : ST_Message;
END_VAR
IF NOT (__ISVALIDREF(_AxisRef)) THEN  MoveVeloBuffer  := E_PROGRESS.PROGRESS_ERROR; RETURN; END_IF
IF NOT bEnable THEN _eState := E_PROGRESS.PROGRESS_INIT; END_IF

CASE _eState
OF
  E_PROGRESS.PROGRESS_INIT:
    IF bEnable 
    THEN
      memset(ADR(_stMsg),0,SIZEOF(_stMsg));
      _nErrorId                     := 0;
      _rValue                       := Velocity;

      _eState                       := E_PROGRESS.PROGRESS_BUSY;

      _stMsg.eType                  := E_MessageType.eMessageVerbose;
      _stMsg.eDevice                := e_Device.Axis + (_AxisRef.NcToPlc.AxisId);
      _stMsg.eSubdevice             := e_SubDevice.fbMoveVelocity1;
      _stMsg.iErrorNumber           := 0;

      _stMsg.sText                  := concat('start : ', TO_STRING(_rValue));

      IF (_MessageLevel = E_MessageType.eMessageVerbose)
      THEN
        f_MessageSet(_stMsg);
      END_IF
    END_IF
END_CASE
CASE _eState
OF
  E_PROGRESS.PROGRESS_BUSY:
    _eState                         := E_PROGRESS.PROGRESS_STARTUP;
    _fbMoveVelocity[1](Axis         := _AxisRef,
                       Execute      := FALSE);

    _fbMoveVelocity[2](Axis         := _AxisRef,
                       Execute      := FALSE);
END_CASE
CASE _eState
OF
  E_PROGRESS.PROGRESS_STARTUP:
    _fbMoveVelocity[1](
                    Axis            := _AxisRef, 
                    Execute         := TRUE,
                    Velocity        := _rValue, 
                    Acceleration    := Acc, 
                    Deceleration    := Dec, 
                    Jerk            := Jerk, 
                    BufferMode      := BufferMode);

    IF _fbMoveVelocity[1].Error
    THEN
      _eState                       := E_PROGRESS.PROGRESS_ERROR;

      _nErrorId                     := _fbMoveVelocity[1].ErrorID;
    
      _stMsg.eType                  := E_MessageType.eMessageError;
      _stMsg.eDevice                := e_Device.Axis + (_AxisRef.NcToPlc.AxisId);
      _stMsg.eSubdevice             :=  e_SubDevice.fbMoveVelocity1;
      _stMsg.iErrorNumber           := _nErrorId;

      _stMsg.sText                  := concat(' : ', TO_STRING(_eState));
    
      f_MessageSet(_stMsg);

    ELSIF (_fbMoveVelocity[1].Busy)
    THEN
      _eState                       := E_PROGRESS.PROGRESS_PREPARE;

      _stMsg.eType                  := E_MessageType.eMessageVerbose;
      _stMsg.eDevice                := e_Device.Axis + (_AxisRef.NcToPlc.AxisId);
      _stMsg.eSubdevice             :=  e_SubDevice.fbMoveVelocity1;
      _stMsg.iErrorNumber           := 0;

      _stMsg.sText                  := concat('FB busy: ', TO_STRING(_eState));

      IF (_MessageLevel = E_MessageType.eMessageVerbose)
      THEN
        f_MessageSet(_stMsg);
      END_IF

    ELSIF (_fbMoveVelocity[1].CommandAborted)
    THEN
      _eState                       := E_PROGRESS.PROGRESS_PREPARE;

      _stMsg.eType                  := E_MessageType.eMessageError;
      _stMsg.eDevice                := e_Device.Axis + (_AxisRef.NcToPlc.AxisId);
      _stMsg.eSubdevice             :=  e_SubDevice.fbMoveVelocity1;
      _stMsg.iErrorNumber           := 0;

      _stMsg.sText                  := concat('FB aborted: ', TO_STRING(_eState));

      f_MessageSet(_stMsg);

    ELSIF (_fbMoveVelocity[1].InVelocity)
    THEN
      _eState                       := E_PROGRESS.PROGRESS_PREPARE;

      _stMsg.eType                  := E_MessageType.eMessageVerbose;
      _stMsg.eDevice                := e_Device.Axis + (_AxisRef.NcToPlc.AxisId);
      _stMsg.eSubdevice             :=  e_SubDevice.fbMoveVelocity1;
      _stMsg.iErrorNumber           := 0;

      _stMsg.sText                  := concat('FB done: ', TO_STRING(_eState));

      IF (_MessageLevel = E_MessageType.eMessageVerbose)
      THEN
        f_MessageSet(_stMsg);
      END_IF
    END_IF
END_CASE
CASE _eState
OF
  E_PROGRESS.PROGRESS_PREPARE:
    _fbMoveVelocity[1](Axis         := _AxisRef);

    IF _fbMoveVelocity[1].Error
    THEN
      _eState                       := E_PROGRESS.PROGRESS_ERROR;

      _nErrorId                     := _fbMoveVelocity[1].ErrorID;
    
      _stMsg.eType                  := E_MessageType.eMessageError;
      _stMsg.eDevice                := e_Device.Axis + (_AxisRef.NcToPlc.AxisId);
      _stMsg.eSubdevice             :=  e_SubDevice.fbMoveVelocity1;
      _stMsg.iErrorNumber           := _nErrorId;

      _stMsg.sText                  := concat(' : ', TO_STRING(_eState));
    
      f_MessageSet(_stMsg);
    
    ELSIF (Velocity <> _rValue)
    THEN
      _eState                       := E_PROGRESS.PROGRESS_CHECK;

      _fbMoveVelocity[1](
                    Axis            := _AxisRef, 
                    Execute         := FALSE);

      _stMsg.eType                  := E_MessageType.eMessageVerbose;
      _stMsg.eDevice                := e_Device.Axis + (_AxisRef.NcToPlc.AxisId);
      _stMsg.eSubdevice             :=  e_SubDevice.fbMoveVelocity2;
      _stMsg.iErrorNumber           := 0;

      _stMsg.sText                  := concat('Velocity changed: ', TO_STRING(_rValue));
      _stMsg.sText                  := concat(_stMsg.sText        , ' to ');
      _stMsg.sText                  := concat(_stMsg.sText        , TO_STRING(Velocity));

      IF (_MessageLevel = E_MessageType.eMessageVerbose)
      THEN
        f_MessageSet(_stMsg);
      END_IF

      _rValue                       := Velocity;
    END_IF
END_CASE
CASE _eState
OF
  E_PROGRESS.PROGRESS_CHECK:
    _fbMoveVelocity[2](
                    Axis            := _AxisRef, 
                    Execute         := TRUE,
                    Velocity        := _rValue, 
                    Acceleration    := Acc, 
                    Deceleration    := Dec, 
                    Jerk            := Jerk, 
                    BufferMode      := BufferMode);

    IF _fbMoveVelocity[2].Error
    THEN
      _eState                       := E_PROGRESS.PROGRESS_ERROR;

      _nErrorId                     := _fbMoveVelocity[2].ErrorID;
    
      _stMsg.eType                  := E_MessageType.eMessageError;
      _stMsg.eDevice                := e_Device.Axis + (_AxisRef.NcToPlc.AxisId);
      _stMsg.eSubdevice             :=  e_SubDevice.fbMoveVelocity2;
      _stMsg.iErrorNumber           := _nErrorId;

      _stMsg.sText                  := concat(' : ', TO_STRING(_eState));
    
      f_MessageSet(_stMsg);

    ELSIF (_fbMoveVelocity[2].Busy)
    THEN
      _eState                       := E_PROGRESS.PROGRESS_PREPARE;

      _stMsg.eType                  := E_MessageType.eMessageVerbose;
      _stMsg.eDevice                := e_Device.Axis + (_AxisRef.NcToPlc.AxisId);
      _stMsg.eSubdevice             :=  e_SubDevice.fbMoveVelocity2;
      _stMsg.iErrorNumber           := 0;

      _stMsg.sText                  := concat('FB busy: ', TO_STRING(_eState));

      IF (_MessageLevel = E_MessageType.eMessageVerbose)
      THEN
        f_MessageSet(_stMsg);
      END_IF

    ELSIF (_fbMoveVelocity[2].CommandAborted)
    THEN
      _eState                       := E_PROGRESS.PROGRESS_PREPARE;

      _stMsg.eType                  := E_MessageType.eMessageError;
      _stMsg.eDevice                := e_Device.Axis + (_AxisRef.NcToPlc.AxisId);
      _stMsg.eSubdevice             :=  e_SubDevice.fbMoveVelocity2;
      _stMsg.iErrorNumber           := 0;

      _stMsg.sText                  := concat('FB aborted: ', TO_STRING(_eState));

      f_MessageSet(_stMsg);

    ELSIF (_fbMoveVelocity[2].InVelocity)
    THEN
      _eState                       := E_PROGRESS.PROGRESS_PREPARE;

      _stMsg.eType                  := E_MessageType.eMessageVerbose;
      _stMsg.eDevice                := e_Device.Axis + (_AxisRef.NcToPlc.AxisId);
      _stMsg.eSubdevice             :=  e_SubDevice.fbMoveVelocity2;
      _stMsg.iErrorNumber           := 0;

      _stMsg.sText                  := concat('FB done: ', TO_STRING(_eState));

      IF (_MessageLevel = E_MessageType.eMessageVerbose)
      THEN
        f_MessageSet(_stMsg);
      END_IF
    END_IF
END_CASE
CASE _eState
OF
  E_PROGRESS.PROGRESS_OCCUPIED:
    _fbMoveVelocity[2](Axis         := _AxisRef);

    IF _fbMoveVelocity[2].Error
    THEN
      _nErrorId                     := _fbMoveVelocity[2].ErrorID;
    
      _stMsg.eType                  := E_MessageType.eMessageError;
      _stMsg.eDevice                := e_Device.Axis + (_AxisRef.NcToPlc.AxisId);
      _stMsg.eSubdevice             :=  e_SubDevice.fbMoveVelocity2;
      _stMsg.iErrorNumber           := _nErrorId;
    
      _stMsg.sText                  := concat(' : ', TO_STRING(_eState));
  
      f_MessageSet(_stMsg);
    
      _eState                       := E_PROGRESS.PROGRESS_ERROR;

    ELSIF (Velocity <> _rValue)
    THEN
      _eState                       := E_PROGRESS.PROGRESS_STARTUP;

      _fbMoveVelocity[2](
                    Axis            := _AxisRef, 
                    Execute         := FALSE);

      _stMsg.eType                  := E_MessageType.eMessageVerbose;
      _stMsg.eDevice                := e_Device.Axis + (_AxisRef.NcToPlc.AxisId);
      _stMsg.eSubdevice             :=  e_SubDevice.fbMoveVelocity1;
      _stMsg.iErrorNumber           := 0;

      _stMsg.sText                  := concat('Velocity changed: ', TO_STRING(_rValue));
      _stMsg.sText                  := concat(_stMsg.sText        , ' to ');
      _stMsg.sText                  := concat(_stMsg.sText        , TO_STRING(Velocity));

      IF (_MessageLevel = E_MessageType.eMessageVerbose)
      THEN
        f_MessageSet(_stMsg);
      END_IF

      _rValue                       := Velocity;
    END_IF
END_CASE
CASE _eState
OF
  E_PROGRESS.PROGRESS_INIT,
  E_PROGRESS.PROGRESS_ERROR:
    _fbMoveVelocity[1](Axis         := _AxisRef,
                       Execute      := FALSE);
    _fbMoveVelocity[2](Axis         := _AxisRef,
                       Execute      := FALSE);
END_CASE


MoveVeloBuffer                      := _eState;
END_METHOD

PROPERTY Override : lreal
GET
Override := _rAxisOverride;
END_GET
SET
_rAxisOverride  := Override;
END_SET
END_PROPERTY

PROPERTY Position : LREAL
GET
Position := _AxisRef.NcToPlc.ActPos;
END_GET
END_PROPERTY

METHOD ReadParameter : E_PROGRESS
VAR_INPUT
  Execute           : BOOL;
  ParameterNumber   : Tc2_MC2.MC_AxisParameter;
END_VAR
VAR_INST
  _eState           : E_PROGRESS;
  _rValue           : LREAL;
  _stMsg            : ST_Message;
END_VAR
IF NOT (__ISVALIDREF(_AxisRef)) THEN  ReadParameter  := E_PROGRESS.PROGRESS_ERROR; RETURN; END_IF
IF NOT Execute THEN _eState := E_PROGRESS.PROGRESS_INIT; END_IF

CASE _eState
OF
  E_PROGRESS.PROGRESS_INIT:
    IF Execute 
    THEN
      memset(ADR(_stMsg),0,SIZEOF(_stMsg));
      _nErrorId                     := 0;
      _rValue                       := 0;
      _eState                       := E_PROGRESS.PROGRESS_BUSY;
    END_IF
END_CASE
CASE _eState
OF
  E_PROGRESS.PROGRESS_BUSY:
    _eState                         := E_PROGRESS.PROGRESS_STARTUP;
    _fbReadParameter(
                    Axis            := _AxisRef, 
                    Enable          := FALSE, 
                    ParameterNumber := ParameterNumber, 
                    ReadMode        := Tc2_MC2.READMODE_ONCE, 
                    Value           => _rValue);
END_CASE
CASE _eState
OF
  E_PROGRESS.PROGRESS_STARTUP:
    _eState                         := E_PROGRESS.PROGRESS_OCCUPIED;
    _fbReadParameter(
                    Axis            := _AxisRef, 
                    Enable          := TRUE, 
                    ParameterNumber := ParameterNumber, 
                    ReadMode        := Tc2_MC2.READMODE_ONCE, 
                    Value           => _rValue);

    _stMsg.eType                    := E_MessageType.eMessageVerbose;
    _stMsg.eDevice                  := e_Device.Axis + (_AxisRef.NcToPlc.AxisId);
    _stMsg.eSubdevice               := e_SubDevice.fbReadParameter;
    _stMsg.iErrorNumber             := 0;

    _stMsg.sText                    := concat(' : ', TO_STRING(_eState));

    IF (_MessageLevel = E_MessageType.eMessageVerbose)
    THEN
      f_MessageSet(_stMsg);
    END_IF
END_CASE
CASE _eState
OF
  E_PROGRESS.PROGRESS_OCCUPIED:
    _fbReadParameter(
                    Axis            := _AxisRef,
                    Value           => _rValue);

    IF (_fbReadParameter.Valid)
    THEN
      _eState                       := E_PROGRESS.PROGRESS_WORKING;
      _rValueParameterRead          := _rValue;
    ELSE
      IF (_fbReadParameter.Error)
      THEN
        _eState                     := E_PROGRESS.PROGRESS_ERROR;
        _nErrorId                   := _fbReadParameter.ErrorID;

        _stMsg.eType                := E_MessageType.eMessageError;
        _stMsg.eDevice              := e_Device.Axis + (_AxisRef.NcToPlc.AxisId);
        _stMsg.eSubdevice           := e_SubDevice.fbReadParameter;
        _stMsg.iErrorNumber         := _nErrorId;

        _stMsg.sText                := concat(' : ', TO_STRING(_eState));

        f_MessageSet(_stMsg);

        _fbReadParameter(
                    Axis            := _AxisRef, 
                    Enable          := FALSE);
      END_IF
    END_IF
END_CASE
CASE _eState
OF
  E_PROGRESS.PROGRESS_WORKING:
    _eState                         := E_PROGRESS.PROGRESS_DONE;
    _fbReadParameter(
                    Axis            := _AxisRef, 
                    Enable          := FALSE);

    _stMsg.eType                    := E_MessageType.eMessageVerbose;
    _stMsg.eDevice                  := e_Device.Axis + (_AxisRef.NcToPlc.AxisId);
    _stMsg.eSubdevice               := e_SubDevice.fbReadParameter;
    _stMsg.iErrorNumber             := 0;

    _stMsg.sText                    := concat(' : ', TO_STRING(_eState));

    IF (_MessageLevel = E_MessageType.eMessageVerbose)
    THEN
      f_MessageSet(_stMsg);
    END_IF
END_CASE

ReadParameter                       := _eState;
END_METHOD

PROPERTY ReadParameterValue : LREAL
GET
ReadParameterValue := _rValueParameterRead;
END_GET
END_PROPERTY

METHOD Reset : E_PROGRESS
VAR_INPUT
  Execute           : BOOL;
END_VAR
VAR_INST
  _eState           : E_PROGRESS;
  _rValue           : LREAL;
  _stMsg            : ST_Message;
END_VAR
IF NOT (__ISVALIDREF(_AxisRef)) THEN  Reset  := E_PROGRESS.PROGRESS_ERROR; RETURN; END_IF
IF NOT Execute THEN _eState := E_PROGRESS.PROGRESS_INIT; END_IF

CASE _eState
OF
  E_PROGRESS.PROGRESS_INIT:
    IF Execute 
    THEN
      memset(ADR(_stMsg),0,SIZEOF(_stMsg));
      _nErrorId                   := 0;
      _rValue                     := 0;
      _eState                     := E_PROGRESS.PROGRESS_BUSY;
    END_IF
END_CASE
CASE _eState
OF
  E_PROGRESS.PROGRESS_BUSY:
    _eState                       := E_PROGRESS.PROGRESS_OCCUPIED;
    _fbReset(
              Axis                := _AxisRef, 
              Execute             := FALSE);
END_CASE
CASE _eState
OF
  E_PROGRESS.PROGRESS_OCCUPIED:
    _fbReset(
              Axis                := _AxisRef, 
              Execute             := TRUE);

    _AxisRef();

    IF _fbReset.Error
    THEN
      _nErrorId                   := _fbReset.ErrorID;

      _stMsg.eType                := E_MessageType.eMessageError;
      _stMsg.eDevice              := e_Device.Axis + (_AxisRef.NcToPlc.AxisId);
      _stMsg.eSubdevice           := e_SubDevice.fbReset;
      _stMsg.iErrorNumber         := _nErrorId;

      f_MessageSet(_stMsg);
      _fbReset(
              Axis                := _AxisRef, 
              Execute             := FALSE);

      _eState                     := E_PROGRESS.PROGRESS_ERROR;
    ELSE
      IF _fbReset.Done OR NOT
         _fbReset.Busy
      THEN
        _eState                   := E_PROGRESS.PROGRESS_WORKING;
      END_IF
    END_IF
END_CASE
CASE _eState
OF
  E_PROGRESS.PROGRESS_WORKING:
    _eState                       := E_PROGRESS.PROGRESS_DONE;
    _fbReset(
              Axis                := _AxisRef, 
              Execute             := FALSE);

    _stMsg.eType                  := E_MessageType.eMessageVerbose;
    _stMsg.eDevice                := e_Device.Axis + (_AxisRef.NcToPlc.AxisId);
    _stMsg.eSubdevice             := e_SubDevice.fbReset;
    _stMsg.iErrorNumber           := 0;

    _stMsg.sText                    := concat(' : ', TO_STRING(_eState));

    IF (_MessageLevel = E_MessageType.eMessageVerbose)
    THEN
      f_MessageSet(_stMsg);
    END_IF
END_CASE


Reset                             := _eState;
END_METHOD

METHOD SendToPos : E_PROGRESS
VAR_INPUT
  Execute         : BOOL;
  Position        : LREAL;
  Distance        : LREAL;
  Vel             : LREAL;
  Acc             : LREAL;
  Dec             : LREAL;
  Jerk            : LREAL;
  BufferMode      : Tc2_MC2.MC_BufferMode;
END_VAR
VAR_INST
  _eState           : E_PROGRESS;
  _rValue           : LREAL;
  _rStart           : LREAL;
  _stMsg            : ST_Message;
END_VAR
IF NOT (__ISVALIDREF(_AxisRef)) THEN  SendToPos  := E_PROGRESS.PROGRESS_ERROR; RETURN; END_IF
IF NOT Execute THEN _eState := E_PROGRESS.PROGRESS_INIT; END_IF

CASE _eState
OF
  E_PROGRESS.PROGRESS_INIT:
    IF Execute 
    THEN
      memset(ADR(_stMsg),0,SIZEOF(_stMsg));
      _nErrorId                     := 0;
      _rValue                       := 0;
      _eState                       := E_PROGRESS.PROGRESS_BUSY;

      _stMsg.eType                  := E_MessageType.eMessageVerbose;
      _stMsg.eDevice                := e_Device.Axis + (_AxisRef.NcToPlc.AxisId);
      _stMsg.eSubdevice             := e_SubDevice.fbSendToPos;
      _stMsg.iErrorNumber           := 0;

      _stMsg.sText                  := concat(' : ', TO_STRING(Position));

      IF (_MessageLevel = E_MessageType.eMessageVerbose)
      THEN
        f_MessageSet(_stMsg);
      END_IF
    END_IF
END_CASE
CASE _eState
OF
  E_PROGRESS.PROGRESS_BUSY:
    _eState                         := E_PROGRESS.PROGRESS_STARTUP;
    _rValue                         := Position;
    _rStart                         := _AxisRef.NcToPlc.ActPos;

    _fbMoveAbsolute[1](Axis         := _AxisRef,
                       Execute      := FALSE);
END_CASE
CASE _eState
OF
  E_PROGRESS.PROGRESS_STARTUP:
    _fbMoveAbsolute[1](
                    Axis            := _AxisRef, 
                    Execute         := TRUE,
                    Position        := _rValue, 
                    Velocity        := Vel, 
                    Acceleration    := Acc, 
                    Deceleration    := Dec, 
                    Jerk            := Jerk, 
                    BufferMode      := BufferMode);

    _rLastTargetPosition            := _fbMoveAbsolute[1].Position;

    _eState                         := E_PROGRESS.PROGRESS_PREPARE;
END_CASE
CASE _eState
OF
  E_PROGRESS.PROGRESS_PREPARE:
    _fbMoveAbsolute[1](Axis         := _AxisRef);

    IF (_fbMoveAbsolute[1].Error)
    THEN
      _nErrorId                     := _fbMoveAbsolute[1].ErrorID;
    
      _stMsg.eType                  := E_MessageType.eMessageError;
      _stMsg.eDevice                := e_Device.Axis + (_AxisRef.NcToPlc.AxisId);
      _stMsg.eSubdevice             :=  e_SubDevice.fbSendToPos;
      _stMsg.iErrorNumber           := _nErrorId;
    
      f_MessageSet(_stMsg);
    
      _eState                         := E_PROGRESS.PROGRESS_ERROR;

    ELSIF (_fbMoveAbsolute[1].Active)
    THEN
      _eState                       := E_PROGRESS.PROGRESS_OCCUPIED;
    END_IF
END_CASE
CASE _eState
OF
  E_PROGRESS.PROGRESS_OCCUPIED:
    _fbMoveAbsolute[1](Axis         := _AxisRef);

    IF (_fbMoveAbsolute[1].Error)
    THEN
      _nErrorId                     := _fbMoveAbsolute[1].ErrorID;
    
      _stMsg.eType                  := E_MessageType.eMessageError;
      _stMsg.eDevice                := e_Device.Axis + (_AxisRef.NcToPlc.AxisId);
      _stMsg.eSubdevice             :=  e_SubDevice.fbSendToPos;
      _stMsg.iErrorNumber           := _nErrorId;
    
      f_MessageSet(_stMsg);
    
      _eState                         := E_PROGRESS.PROGRESS_ERROR;

    ELSIF (_AxisRef.NcToPlc.ActPos > _rStart + Distance)
    THEN
      _fbMoveAbsolute[1](Axis       := _AxisRef,
                         Execute    := FALSE);

      _eState                       := E_PROGRESS.PROGRESS_DONE;

      _stMsg.eType                  := E_MessageType.eMessageVerbose;
      _stMsg.eDevice                := e_Device.Axis + (_AxisRef.NcToPlc.AxisId);
      _stMsg.eSubdevice             := e_SubDevice.fbSendToPos;
      _stMsg.iErrorNumber           := 0;

      _stMsg.sText                  := concat(' : ', TO_STRING(_eState));

      IF (_MessageLevel = E_MessageType.eMessageVerbose)
      THEN
        f_MessageSet(_stMsg);
      END_IF
    END_IF
END_CASE

SendToPos                             := _eState;
END_METHOD

METHOD StartUp : E_PROGRESS
VAR_INPUT
  Execute           : BOOL;
END_VAR
VAR_INST
  _eState           : E_PROGRESS;
  _uiEncType        : UDINT;

  _sEncoder,
  _sName            : STRING(30);

  _rValue           : LREAL;
  _stMsg            : ST_Message;
END_VAR
IF NOT (__ISVALIDREF(_AxisRef)) THEN  StartUp  := E_PROGRESS.PROGRESS_ERROR; RETURN; END_IF
IF NOT Execute THEN _eState := E_PROGRESS.PROGRESS_INIT; END_IF


